METHOD An_unrecognized_version_is_reported_once_with_its_owner
TEST('An_unrecognized_version_is_reported_once_with_its_owner');
_M_Arm();
_M_TakeLoss();
_version := 7;                            // a real image, written by another layout
AssertFalse(Condition := _u.Child.M_RestoreStationCfg(pVersion := ADR(_version),
    SchemaVersion := 1),
    Message := 'an unrecognized image is REJECTED, never read by field position');
AssertEquals_UINT(Expected := 1, Actual := _version,
    Message := 'the version is stamped forward so the loss annunciates once, not every boot');
AssertTrue(Condition := _M_TakeLoss(),
    Message := 'losing a real image is reported (3.8b: never silent)');
AssertEquals_STRING(Expected := 'Test.Durability.Child', Actual := _path,
    Message := 'the report names the OWNING module, which is what makes it actionable');
AssertEquals_UINT(Expected := 1, Actual := _expected,
    Message := 'the report carries the schema this build understands');
AssertEquals_UINT(Expected := 7, Actual := _found,
    Message := 'and the schema actually found');
AssertFalse(Condition := _M_TakeLoss(),
    Message := 'taking a loss clears it: one annunciation per boot, not one per scan');
TEST_FINISHED();
END_METHOD

// §3.8b: the annunciation is AUTO_RESET and therefore never blocking. The
// consequence belongs to E_ConfigRestorePolicy, so a station that declared
// DEFAULTS_AND_ANNUNCIATE really does keep running while the alarm stands.
METHOD The_root_annunciates_a_loss_without_blocking_on_its_own
TEST('The_root_annunciates_a_loss_without_blocking_on_its_own');
_M_Arm();
_M_TakeLoss();
_u.SetConfigRestorePolicy(Policy := E_ConfigRestorePolicy.DEFAULTS_AND_ANNUNCIATE);
_version := 9;
_u.Child.M_RestoreStationCfg(pVersion := ADR(_version), SchemaVersion := 1);
_u();                                     // OnCyclic drains and annunciates
AssertTrue(Condition := _u.ConfigPersist.RestoreLost,
    Message := 'the root publishes that something in its subtree lost its image');
AssertEquals_STRING(Expected := 'Test.Durability.Child',
    Actual := _u.ConfigPersist.LostPath,
    Message := 'and publishes whose');
AssertFalse(Condition := _u.ConfigPersist.RestoreAcknowledged,
    Message := 'nobody has accepted the loss yet');
AssertFalse(Condition := _u.AlarmLog.Blocking,
    Message := 'the standing annunciation is AUTO_RESET: loud, never a Start block');
_released := _u.ReleaseReportStart(Report := _report);
AssertTrue(Condition := _released,
    Message := 'DEFAULTS_AND_ANNUNCIATE runs the station and lets the alarm stand');
TEST_FINISHED();
END_METHOD

// §3.8b BLOCK_UNTIL_ACKNOWLEDGED: no START_STOP release until an operator of at
// least ENGINEER level accepts the loss. The release is restored by the
// ACKNOWLEDGEMENT, never by the loss going away - nothing brings a lost image back.
METHOD Blocking_policy_refuses_start_until_an_engineer_acknowledges
TEST('Blocking_policy_refuses_start_until_an_engineer_acknowledges');
_M_Arm();
_M_TakeLoss();
_u.SetConfigRestorePolicy(Policy := E_ConfigRestorePolicy.BLOCK_UNTIL_ACKNOWLEDGED);
_version := 11;
_u.Child.M_RestoreStationCfg(pVersion := ADR(_version), SchemaVersion := 1);
_u();
AssertTrue(Condition := _u.ConfigPersist.RestoreLost,
    Message := 'the loss is published');
_released := _u.ReleaseReportStart(Report := _report);
AssertFalse(Condition := _released,
    Message := 'a station that lost its commissioning does not start pretending it did not');
AssertFalse(Condition := _u.Start(),
    Message := 'and Start consumes that same report, so the two cannot disagree');
// An operator below ENGINEER cannot make this go away. A login or logout is a
// REQUEST that Access.Cyclic applies on the Unit's next call, so each is followed
// by one - without it the level asserted against was simply the previous one.
_u.Access.RequestLogout();
_u();
AssertFalse(Condition := _u.AcknowledgeConfigRestore(),
    Message := 'acknowledging a lost commissioning is an ENGINEER-level act (3.8b)');
AssertFalse(Condition := _u.ConfigPersist.RestoreAcknowledged,
    Message := 'a refused acknowledgement changes nothing');
AssertTrue(Condition := _u.Access.RequestLogin(User := 'eng', Secret := '4242'),
    Message := 'the fixture provides an ENGINEER session');
_u();
AssertTrue(Condition := _u.AcknowledgeConfigRestore(),
    Message := 'an ENGINEER may accept the loss');
_released := _u.ReleaseReportStart(Report := _report);
AssertTrue(Condition := _released,
    Message := 'the acknowledgement, not the condition, is what releases Start again');
AssertTrue(Condition := _u.ConfigPersist.RestoreLost,
    Message := 'and the loss itself is still published: acknowledged is not undone');
_u.Access.RequestLogout();
_u.SetConfigRestorePolicy(Policy := E_ConfigRestorePolicy.DEFAULTS_AND_ANNUNCIATE);
TEST_FINISHED();
END_METHOD

// §3.8b: "Transport acknowledgement and Accepted mean a value is LIVE, not that
// it is DURABLE." This is that sentence as a test.
METHOD An_accepted_write_is_pending_until_the_store_completes
TEST('An_accepted_write_is_pending_until_the_store_completes');
_M_Arm();
_u.SetConfigPersistWindow(WindowMs := 60000);
_persist.M_SetOutcome(Failed := FALSE, Refuse := FALSE);
_persist.M_SetHold(Hold := TRUE);         // the store does not finish yet
AssertTrue(Condition := _u.WriteConfig(TargetPath := 'Test.Durability',
    WriteKey := 'probe.cycleLimit', Revision := 1, TextValue := '42'),
    Message := 'the write is accepted');
AssertTrue(Condition := _u.ConfigPersist.Pending,
    Message := 'accepted means LIVE - the root publishes that it is not yet durable');
AssertFalse(Condition := _u.ConfigPersist.Failed,
    Message := 'pending is not failed');
_u();
AssertTrue(Condition := _u.ConfigPersist.Pending,
    Message := 'and it stays pending for as long as the store is still working');
_persist.M_SetHold(Hold := FALSE);
_u();
_u();
AssertFalse(Condition := _u.ConfigPersist.Pending,
    Message := 'the value is durable once the store completes');
AssertFalse(Condition := _u.ConfigPersist.Failed,
    Message := 'a completed write is not a failed one');
TEST_FINISHED();
END_METHOD

METHOD A_store_that_refuses_publishes_PersistFailed
TEST('A_store_that_refuses_publishes_PersistFailed');
_M_Arm();
_u.SetConfigPersistWindow(WindowMs := 60000);
_persist.M_SetHold(Hold := FALSE);
_persist.M_SetOutcome(Failed := FALSE, Refuse := TRUE);
AssertTrue(Condition := _u.WriteConfig(TargetPath := 'Test.Durability',
    WriteKey := 'probe.cycleLimit', Revision := 1, TextValue := '43'),
    Message := 'the VALUE is still accepted: it is live, and that is not in doubt');
AssertTrue(Condition := _u.ConfigPersist.Failed,
    Message := 'a store that will not even start is a failure, not a quiet no-op');
AssertTrue(Condition := _u.ConfigPersist.Pending,
    Message := 'and the value is STILL not durable, so it stays pending');
AssertFalse(Condition := _u.AlarmLog.Blocking,
    Message := 'the annunciation does not stop a machine that can still finish its parts');
// A store that starts working again clears both on the next accepted write.
_persist.M_SetOutcome(Failed := FALSE, Refuse := FALSE);
AssertTrue(Condition := _u.WriteConfig(TargetPath := 'Test.Durability',
    WriteKey := 'probe.cycleLimit', Revision := 1, TextValue := '44'),
    Message := 'a later write is accepted');
_u();
_u();
AssertFalse(Condition := _u.ConfigPersist.Failed,
    Message := 'a successful write clears the failure it re-armed');
TEST_FINISHED();
END_METHOD

// §3.8b declares a BOUNDED window, and a bound nobody measures is not a bound.
// WindowMs := 0 declares "durable in the same scan or not at all", which is the
// honest declaration for a store that cannot be slow.
METHOD An_elapsed_window_publishes_PersistFailed
TEST('An_elapsed_window_publishes_PersistFailed');
_M_Arm();
IF NOT _winArmed THEN
    _winArmed := TRUE;
    _persist.M_SetOutcome(Failed := FALSE, Refuse := FALSE);
    _persist.M_SetHold(Hold := TRUE);     // never completes
    _u.SetConfigPersistWindow(WindowMs := 0);
    AssertTrue(Condition := _u.WriteConfig(TargetPath := 'Test.Durability',
        WriteKey := 'probe.cycleLimit', Revision := 1, TextValue := '45'),
        Message := 'the write is accepted');
    AssertTrue(Condition := _u.ConfigPersist.Pending, Message := 'and is pending');
    RETURN;                               // the window is measured in TIME(), which
END_IF                                    // does not advance inside one scan
_u();
_winScans := _winScans + 1;
IF NOT _u.ConfigPersist.Failed AND (_winScans < 50) THEN
    RETURN;                               // bounded: 50 scans, far past a 0 ms window
END_IF
AssertTrue(Condition := _u.ConfigPersist.Failed,
    Message := 'a store still working past the DECLARED window has failed the declaration');
AssertTrue(Condition := _u.ConfigPersist.Pending,
    Message := 'the value is still not durable, so it is still pending');
_persist.M_SetHold(Hold := FALSE);
_u.SetConfigPersistWindow(WindowMs := PL_Fraktal.CONFIG_PERSIST_WINDOW_MS);
_u();
TEST_FINISHED();
END_METHOD

END_FUNCTION_BLOCK

// ---- Fraktal_Tests/FB_ConfigSet_Tests.TcPOU
// Core §3.8b under test, the half that is about CONTENT:
//
//   * a set is a PROJECTION of the same deterministic walk that builds the
//     §3.10.2 manifest - not a second list of what a station's configuration
//     consists of, which would be free to drift from the first;
//   * it is records keyed by (Scope, WriteKey), never a byte image, which is
//     what lets one bad value be rejected without rejecting all of them;
//   * a load is STAGED and ALL-OR-NOTHING, so a set that is wrong anywhere
//     changes nothing anywhere;
//   * and the whole set moves as TEXT, because a set that cannot leave the
//     controller is just retentive memory with a name on it.
FUNCTION_BLOCK FB_ConfigSet_Tests EXTENDS TcUnit.FB_TestSuite
VAR
    _u       : FB_ProbeConfigUnit;
    _init    : BOOL;
    // PL_Fraktal.MAX_CONFIG_SETS is 4 and the store never evicts a set, so every
    // DELIBERATELY WRONG import shares the one name 'imported' (each overwrites
    // the last). Seven distinct names filled the store by the fifth test, and the
    // later imports were refused as 'full' before reaching the rule they test.
    _store   : FB_LocalConfigStore;
    _json    : FB_ConfigSetJson;
    _pager   : FB_ConfigPager;
    _page    : ST_ConfigPage;
    _info    : ST_ConfigSetInfo;
    _record  : ST_ConfigRecord;
    _decoded : ST_ConfigRecord;
    _line    : STRING(480);
    _i       : INT;
    _capabilities : INT;
    // A whole Unit is far too large for a method local: as one it put ~330 KB on a
    // 48 KB task stack (C0297) and the suite could never run. It lives here instead.
    _bare     : FB_ProbeConfigUnit;
    _bareInit : BOOL;
END_VAR

A_saved_set_is_the_manifest_walk_projected();
A_set_round_trips_through_the_store();
Loading_a_set_restores_every_value_it_carries();
One_bad_record_aborts_the_whole_load_and_names_it();
A_capability_that_no_longer_exists_is_reported_not_dropped();
A_set_from_another_root_is_refused();
A_record_round_trips_through_its_json_line();
A_malformed_json_line_is_refused_whole();
A_model_set_is_not_applied_as_per_field_writes();
Set_operations_need_a_store_and_the_CONFIG_SET_gate();
A_deleted_set_is_gone_and_frees_its_slot();
A_line_longer_than_a_request_imports_in_pieces();

// One-time wiring. Nothing here is persistence-specific: a store is injected
// exactly as a composition root injects it, and every value in the resulting
// sets came from an ordinary M_RegisterConfig* call on the probes.
METHOD PRIVATE _M_Arm
IF _init THEN
    RETURN;
END_IF
_init := TRUE;
_u.Setup(Name := 'Test.CfgSet');
_u();
_u.SetConfigStore(Store := _store);
// The store is PERSISTENT, so it still holds whatever the previous run saved:
// start every run from an empty store, through the same delete a station has.
FOR _i := 1 TO PL_Fraktal.MAX_CONFIG_SETS DO
    IF NOT _store.M_InfoAt(Index := 1, Info := _info) THEN
        EXIT;
    END_IF
    _u.DeleteConfigSet(SetName := _info.SetName);
END_FOR
END_METHOD

// Count the writable STATION_CFG capabilities the MANIFEST publishes, by walking
// it exactly as a client does. The set has to contain the same number - that
// equality is what "a set is a projection of the same walk" means in practice.
METHOD PRIVATE _M_CountStationCapabilities : INT
VAR
    page  : INT;
    i     : INT;
    pages : INT;
END_VAR
_M_CountStationCapabilities := 0;
pages := 1;
FOR page := 0 TO 63 DO
    IF page >= pages THEN
        RETURN;
    END_IF
    _pager.M_Setup(Target := ADR(_page), PageIndex := page, Revision := 1);
    _u.M_AppendConfig(Pager := _pager);
    _pager.M_Finish();
    pages := _page.PageCount;
    FOR i := 1 TO _page.EntryCount DO
        IF _page.Entries[i].Writable THEN
            IF _page.Entries[i].ConfigKind = E_ConfigKind.STATION_CFG THEN
                _M_CountStationCapabilities := _M_CountStationCapabilities + 1;
            END_IF
        END_IF
    END_FOR
END_FOR
END_METHOD

// Push one JSON line into the store through the ordinary import route, so a
// suite can build a DELIBERATELY WRONG set the same way a foreign tool would.
METHOD PRIVATE _M_Import : BOOL
VAR_INPUT
    Line   : STRING(480);
    Commit : BOOL;
END_VAR
_M_Import := _u.ImportConfigSetLine(Line := Line, Commit := Commit);
END_METHOD

METHOD A_saved_set_is_the_manifest_walk_projected
TEST('A_saved_set_is_the_manifest_walk_projected');
_M_Arm();
_capabilities := _M_CountStationCapabilities();
AssertTrue(Condition := _capabilities > 0,
    Message := 'the fixture publishes STATION_CFG capabilities to project');
AssertTrue(Condition := _u.SaveConfigSet(SetName := 'baseline',
    Kind := E_ConfigKind.STATION_CFG),
    Message := 'a station set saves');
AssertTrue(Condition := _store.M_ReadInfo(SetName := 'baseline', Info := _info),
    Message := 'and is readable back out of the store');
AssertEquals_INT(Expected := _capabilities, Actual := _info.RecordCount,
    Message := 'the set contains exactly the capabilities the manifest publishes - one walk, not two');
AssertEquals_STRING(Expected := 'Test.CfgSet', Actual := _info.RootIdentity,
    Message := 'a set carries the identity of the root that produced it');
AssertTrue(Condition := _info.ConfigRev > 0,
    Message := 'and the ConfigRev it was taken at');
TEST_FINISHED();
END_METHOD

METHOD A_set_round_trips_through_the_store
TEST('A_set_round_trips_through_the_store');
_M_Arm();
_u.SaveConfigSet(SetName := 'baseline', Kind := E_ConfigKind.STATION_CFG);
AssertTrue(Condition := _store.M_ReadInfo(SetName := 'baseline', Info := _info),
    Message := 'the header reads back');
AssertTrue(Condition := _store.M_ReadRecord(SetName := 'baseline', Index := 1,
    Record := _record), Message := 'and so does record 1');
AssertTrue(Condition := _record.WriteKey <> '',
    Message := 'every record carries the mutation identity it will be replayed through');
AssertFalse(Condition := _store.M_ReadRecord(SetName := 'baseline',
    Index := _info.RecordCount + 1, Record := _record),
    Message := 'reading past the end is refused, not clamped');
AssertFalse(Condition := _store.M_ReadInfo(SetName := 'nosuchset', Info := _info),
    Message := 'an absent set is absent, not empty');
AssertTrue(Condition := _u.ListConfigSets(),
    Message := 'the listing is served');
AssertTrue(Condition := _u.ConfigSetCount >= 1,
    Message := 'and shows the set that was just saved');
TEST_FINISHED();
END_METHOD

METHOD Loading_a_set_restores_every_value_it_carries
TEST('Loading_a_set_restores_every_value_it_carries');
_M_Arm();
_u.WriteConfig(TargetPath := 'Test.CfgSet', WriteKey := 'probe.cycleLimit',
    Revision := 1, TextValue := '250');
AssertTrue(Condition := _u.SaveConfigSet(SetName := 'commissioned',
    Kind := E_ConfigKind.STATION_CFG), Message := 'save the commissioned state');
// Somebody then changes the machine.
_u.WriteConfig(TargetPath := 'Test.CfgSet', WriteKey := 'probe.cycleLimit',
    Revision := 1, TextValue := '7');
AssertEquals_DINT(Expected := 7, Actual := _u.CycleLimit,
    Message := 'the live value really changed');
AssertTrue(Condition := _u.LoadConfigSet(SetName := 'commissioned'),
    Message := 'the saved set loads');
AssertEquals_DINT(Expected := 250, Actual := _u.CycleLimit,
    Message := 'and the commissioned value is back, replayed through the owning handler');
TEST_FINISHED();
END_METHOD

// §3.8b: "one rejection aborts the whole load naming the offending
// (Scope, WriteKey)" and "a half-applied machine parametrization is never a
// valid outcome". The set below is valid in every record but one.
METHOD One_bad_record_aborts_the_whole_load_and_names_it
TEST('One_bad_record_aborts_the_whole_load_and_names_it');
_M_Arm();
_u.WriteConfig(TargetPath := 'Test.CfgSet', WriteKey := 'probe.cycleLimit',
    Revision := 1, TextValue := '99');
// A set whose FIRST record is fine and whose SECOND is out of the declared
// range - built as text, exactly as a foreign tool or a hand edit would.
AssertTrue(Condition := _M_Import(Line :=
    '{"set":"imported","root":"Test.CfgSet","schema":1,"configRev":1,"kind":1,"model":"","records":2,"created":0,"clock":0}',
    Commit := FALSE), Message := 'the header opens the import');
AssertTrue(Condition := _M_Import(Line :=
    '{"scope":"Test.CfgSet.Child","key":"probe.retries","rev":1,"kind":1,"type":0,"value":"4"}',
    Commit := FALSE), Message := 'a good record is taken');
AssertTrue(Condition := _M_Import(Line :=
    '{"scope":"Test.CfgSet","key":"probe.cycleLimit","rev":1,"kind":1,"type":0,"value":"99999"}',
    Commit := TRUE), Message := 'and so is the out-of-range one: the STORE does not validate');
AssertFalse(Condition := _u.LoadConfigSet(SetName := 'imported'),
    Message := 'the LOAD validates, and one bad record refuses the whole set');
AssertEquals_DINT(Expected := 99, Actual := _u.CycleLimit,
    Message := 'nothing was applied - not even the record that came BEFORE the bad one');
AssertEquals_DINT(Expected := 3, Actual := _u.Child.Retries,
    Message := 'and not the good record in another module either');
AssertEquals_STRING(Expected := 'Test.CfgSet',
    Actual := _u.ConfigPersist.LastRejectScope,
    Message := 'the refusal names the scope of the offending record');
AssertEquals_STRING(Expected := 'probe.cycleLimit',
    Actual := _u.ConfigPersist.LastRejectKey,
    Message := 'and its write key');
TEST_FINISHED();
END_METHOD

// §3.8b: "Records whose capability no longer exists in the target are reported,
// never silently dropped." A set that quietly skipped the one value that
// mattered would restore a machine to ALMOST its commissioned state, which is
// the failure that is hardest to notice.
METHOD A_capability_that_no_longer_exists_is_reported_not_dropped
TEST('A_capability_that_no_longer_exists_is_reported_not_dropped');
_M_Arm();
_M_Import(Line :=
    '{"set":"imported","root":"Test.CfgSet","schema":1,"configRev":1,"kind":1,"model":"","records":1,"created":0,"clock":0}',
    Commit := FALSE);
_M_Import(Line :=
    '{"scope":"Test.CfgSet","key":"probe.valueThatWasRemoved","rev":1,"kind":1,"type":0,"value":"1"}',
    Commit := TRUE);
AssertFalse(Condition := _u.LoadConfigSet(SetName := 'imported'),
    Message := 'a record nothing owns any more refuses the load');
AssertEquals_STRING(Expected := 'probe.valueThatWasRemoved',
    Actual := _u.ConfigPersist.LastRejectKey,
    Message := 'and is REPORTED by name rather than passed over');
TEST_FINISHED();
END_METHOD

METHOD A_set_from_another_root_is_refused
TEST('A_set_from_another_root_is_refused');
_M_Arm();
_M_Import(Line :=
    '{"set":"imported","root":"SomeOtherPress","schema":1,"configRev":1,"kind":1,"model":"","records":1,"created":0,"clock":0}',
    Commit := FALSE);
_M_Import(Line :=
    '{"scope":"SomeOtherPress","key":"probe.cycleLimit","rev":1,"kind":1,"type":0,"value":"5"}',
    Commit := TRUE);
AssertFalse(Condition := _u.LoadConfigSet(SetName := 'imported'),
    Message := 'a set carries the identity of the root that produced it so this can be asked');
AssertEquals_STRING(Expected := 'SomeOtherPress',
    Actual := _u.ConfigPersist.LastRejectScope,
    Message := 'and the refusal names the root it actually came from');
TEST_FINISHED();
END_METHOD

// A set that cannot leave the controller is retentive memory with a name on it.
// One JSON object per record is what makes it movable - and keeps every value
// independently identified and independently rejectable, which is exactly the
// property §3.8b says a byte image loses.
METHOD A_record_round_trips_through_its_json_line
TEST('A_record_round_trips_through_its_json_line');
_M_Arm();
_record.Scope := 'Test.CfgSet.Child';
_record.WriteKey := 'probe.label';
_record.Revision := 2;
_record.Kind := E_ConfigKind.STATION_CFG;
_record.ValueType := E_ConfigValueType.TEXT;
_record.ValueText := 'a "quoted" value';   // the two characters JSON must escape
_line := _json.M_Record(Record := _record);
AssertTrue(Condition := _line <> '',
    Message := 'a valid record renders');
AssertTrue(Condition := _json.M_ParseRecord(Line := _line, Record := _decoded),
    Message := 'and parses back');
AssertEquals_STRING(Expected := 'Test.CfgSet.Child', Actual := _decoded.Scope,
    Message := 'the owning scope survives the round trip');
AssertEquals_STRING(Expected := 'probe.label', Actual := _decoded.WriteKey,
    Message := 'so does the mutation identity');
AssertEquals_STRING(Expected := 'a "quoted" value', Actual := _decoded.ValueText,
    Message := 'and so does a value containing the delimiter itself');
AssertEquals_UDINT(Expected := 2, Actual := _decoded.Revision,
    Message := 'the capability revision travels with the record, so a load can reject a value whose meaning changed');
TEST_FINISHED();
END_METHOD

METHOD A_malformed_json_line_is_refused_whole
TEST('A_malformed_json_line_is_refused_whole');
_M_Arm();
_decoded.WriteKey := 'untouched';
AssertFalse(Condition := _json.M_ParseRecord(
    Line := '{"scope":"x","key":"y","rev":1,"kind":1,"type":0', Record := _decoded),
    Message := 'a truncated line is not a record');
AssertFalse(Condition := _json.M_ParseRecord(
    Line := '{"scope":"x","key":"y","rev":"notanumber","kind":1,"type":0,"value":"1"}',
    Record := _decoded), Message := 'nor is one whose revision is not a number');
AssertFalse(Condition := _json.M_ParseRecord(
    Line := '{"scope":"x","key":"y","rev":1,"kind":9,"type":0,"value":"1"}',
    Record := _decoded), Message := 'nor one whose kind is outside E_ConfigKind');
AssertEquals_STRING(Expected := 'untouched', Actual := _decoded.WriteKey,
    Message := 'a refused line leaves the caller record exactly as it was');
AssertFalse(Condition := _json.M_ParseHeader(
    Line := '{"scope":"x","key":"y","rev":1,"kind":1,"type":0,"value":"1"}',
    Info := _info), Message := 'a record line is not a header, and says so');
TEST_FINISHED();
END_METHOD

// §3.8b: a MODEL set "shall be applied through the §3.8 changeover transaction
// ... never as a sequence of per-field writes". Replaying it here would be
// exactly that forbidden sequence, so it is refused. Saving one is supported;
// loading one is a changeover this build does not implement, and refusing is
// the honest half of that.
METHOD A_model_set_is_not_applied_as_per_field_writes
TEST('A_model_set_is_not_applied_as_per_field_writes');
_M_Arm();
_M_Import(Line :=
    '{"set":"imported","root":"Test.CfgSet","schema":1,"configRev":1,"kind":0,"model":"ALU","records":1,"created":0,"clock":0}',
    Commit := FALSE);
_M_Import(Line :=
    '{"scope":"Test.CfgSet","key":"probe.cycleLimit","rev":1,"kind":0,"type":0,"value":"12"}',
    Commit := TRUE);
AssertFalse(Condition := _u.LoadConfigSet(SetName := 'imported'),
    Message := 'a model set is not replayed as per-field writes');
AssertEquals_STRING(Expected := 'ALU', Actual := _u.ConfigPersist.LastRejectScope,
    Message := 'and the refusal names the model it was for');
TEST_FINISHED();
END_METHOD

// §3.8b/§7.7: saving, loading or importing a SET is the separate gated action
// CONFIG_SET, "because replacing a machine's entire parametrization is not the
// same decision as changing one number". And a root with no store offers the
// operations not at all rather than failing when somebody finally tries.
METHOD Set_operations_need_a_store_and_the_CONFIG_SET_gate
TEST('Set_operations_need_a_store_and_the_CONFIG_SET_gate');
_M_Arm();
IF NOT _bareInit THEN
    _bareInit := TRUE;
    _bare.Setup(Name := 'Test.NoStore');   // registers once, like any root
END_IF
_bare();
AssertFalse(Condition := _bare.ConfigPersist.StorePresent,
    Message := 'a root with no store says so, rather than pretending');
AssertFalse(Condition := _bare.SaveConfigSet(SetName := 'x',
    Kind := E_ConfigKind.STATION_CFG),
    Message := 'and refuses to save');
AssertFalse(Condition := _bare.LoadConfigSet(SetName := 'x'),
    Message := 'and to load');
AssertTrue(Condition := _u.ConfigPersist.StorePresent,
    Message := 'a wired root publishes that sets are available');
AssertEquals_DINT(Expected := TO_DINT(E_ConfigStore.LOCAL_RETAIN),
    Actual := TO_DINT(_u.ConfigPersist.StoreKind),
    Message := 'and publishes WHERE they live, so a saved set is not taken on faith');
AssertTrue(Condition := _u.Access.RequestLogout(),
    Message := 'no session is required by the shipped fully-open policy');
AssertTrue(Condition := _u.SaveConfigSet(SetName := 'open',
    Kind := E_ConfigKind.STATION_CFG),
    Message := 'so an open station saves without a login - access control is never a silent lock-in');
TEST_FINISHED();
END_METHOD

// §3.8b round trip. An exported line may hold 480 characters but a request
// carries 255, so a long record arrives in pieces (IMPORT_CONFIG_SET with
// IntValue = 1). Without the join, a station's own export could not come back.
METHOD A_line_longer_than_a_request_imports_in_pieces
VAR
    header : STRING(480);
    first  : STRING(255);
    rest   : STRING(255);
    k      : INT;
    size   : INT;                          // measured by scanning, not by LEN
    p      : POINTER TO BYTE;
END_VAR
TEST('A_line_longer_than_a_request_imports_in_pieces');
_M_Arm();
// The previous test leaves the store full: free a slot, then reuse fill2's
// header so the import overwrites a set this suite owns.
_u.DeleteConfigSet(SetName := 'fill1');
_u.ExportConfigSetLine(SetName := 'fill2', Line := 0);
header := _u.ConfigSetDocument;
AssertTrue(Condition := header <> '', Message := 'a header to import under');
_record.Scope := 'Test.CfgSet.Child.Long';
_record.WriteKey := '';
FOR k := 1 TO 14 DO
    _record.WriteKey := CONCAT(_record.WriteKey, 'probe.long');
END_FOR
_record.Revision := 1;
_record.Kind := E_ConfigKind.STATION_CFG;
_record.ValueType := E_ConfigValueType.TEXT;
_record.ValueText := '';
FOR k := 1 TO 7 DO
    _record.ValueText := CONCAT(_record.ValueText, '0123456789');
END_FOR
_line := _json.M_Record(Record := _record);
// The length is measured by scanning to the terminator, independently of LEN:
// the standard string functions are specified to 255 characters, so neither
// LEN nor CONCAT may be trusted past it without proof.
size := 0;
p := ADR(_line);
WHILE size < 480 AND p^ <> 0 DO
    size := size + 1;
    p := p + 1;
END_WHILE
AssertTrue(Condition := size > 255,
    Message := CONCAT('the record renders past 255 characters; scanned ', INT_TO_STRING(size)));
// Measured on the runtime (2026-09-28): LEN reported 255 for this 290-character
// line. That is why the codec scans instead, and why this test does too.
AssertTrue(Condition := _json.M_ParseRecord(Line := _line, Record := _decoded),
    Message := 'the long line is whole: it parses back');
AssertEquals_STRING(Expected := _record.ValueText, Actual := _decoded.ValueText,
    Message := 'and its value is intact, so rendering did not truncate');
// Pieces by byte copy, so the test does not depend on LEFT/MID past 255.
MEMSET(ADR(first), 0, SIZEOF(first));
MEMSET(ADR(rest), 0, SIZEOF(rest));
MEMCPY(ADR(first), ADR(_line), 200);
IF size > 200 THEN
    MEMCPY(ADR(rest), ADR(_line) + 200, TO_UDINT(MIN(size - 200, 255)));
END_IF
AssertTrue(Condition := _M_Import(Line := header, Commit := FALSE),
    Message := 'the header opens the import');
AssertTrue(Condition := _u.ImportConfigSetPiece(Piece := first, More := TRUE,
    Commit := FALSE), Message := 'the first piece is held');
AssertTrue(Condition := _u.ImportConfigSetPiece(Piece := rest, More := FALSE,
    Commit := TRUE), Message := 'the last piece completes the line, which imports and commits');
AssertTrue(Condition := _store.M_ReadRecord(SetName := 'fill2', Index := 1,
    Record := _decoded), Message := 'the joined record is in the store');
AssertEquals_STRING(Expected := _record.ValueText, Actual := _decoded.ValueText,
    Message := 'and its value arrived whole, not truncated at 255');
AssertEquals_STRING(Expected := _record.WriteKey, Actual := _decoded.WriteKey,
    Message := 'as did its 140-character key');
// Refused, never truncated: pieces that would exceed the line width.
AssertTrue(Condition := _u.ImportConfigSetPiece(Piece := first, More := TRUE,
    Commit := FALSE), Message := 'a piece is held');
AssertTrue(Condition := _u.ImportConfigSetPiece(Piece := first, More := TRUE,
    Commit := FALSE), Message := 'and a second (400 characters so far)');
AssertFalse(Condition := _u.ImportConfigSetPiece(Piece := first, More := FALSE,
    Commit := FALSE), Message := 'a join past 480 characters is refused');
TEST_FINISHED();
END_METHOD

// §3.8b: without a delete, a store that has held MAX_CONFIG_SETS names can
// only ever overwrite one of them again - a new product's recipe could not be
// kept without destroying an old one under its name.
METHOD A_deleted_set_is_gone_and_frees_its_slot
VAR
    fill : STRING(80);
END_VAR
TEST('A_deleted_set_is_gone_and_frees_its_slot');
_M_Arm();
// The earlier tests leave the store full, so start from empty: this test is
// about what delete does, not about which sets happened to be there.
FOR _i := 1 TO PL_Fraktal.MAX_CONFIG_SETS DO
    IF NOT _store.M_InfoAt(Index := 1, Info := _info) THEN
        EXIT;
    END_IF
    _u.DeleteConfigSet(SetName := _info.SetName);
END_FOR
AssertTrue(Condition := _u.SaveConfigSet(SetName := 'scratch',
    Kind := E_ConfigKind.STATION_CFG), Message := 'a set to delete is saved');
AssertTrue(Condition := _u.DeleteConfigSet(SetName := 'scratch'),
    Message := 'an existing set is deleted');
AssertFalse(Condition := _store.M_ReadInfo(SetName := 'scratch', Info := _info),
    Message := 'and is no longer readable');
AssertFalse(Condition := _u.DeleteConfigSet(SetName := 'scratch'),
    Message := 'deleting what is not there is refused, not silently accepted');
AssertTrue(Condition := _u.ConfigPersist.Pending,
    Message := 'a delete changes retained memory, so it is not durable until written out');
AssertEquals_INT(Expected := 0, Actual := _store.M_Count(),
    Message := 'every set can be removed');
// The freed slots are usable: fill the store to capacity under fresh names.
FOR _i := 1 TO PL_Fraktal.MAX_CONFIG_SETS DO
    fill := CONCAT('fill', INT_TO_STRING(_i));
    AssertTrue(Condition := _u.SaveConfigSet(SetName := fill,
        Kind := E_ConfigKind.STATION_CFG), Message := 'each freed slot takes a new name');
END_FOR
TEST_FINISHED();
END_METHOD

END_FUNCTION_BLOCK

// ---- Fraktal_Tests/FB_DataClass_Tests.TcPOU
// Core §3.8d under test: data classes and raise-only per-value access.
// Every test body is guarded: TcUnit calls finished tests every scan, and these
// write to one shared probe.
FUNCTION_BLOCK FB_DataClass_Tests EXTENDS TcUnit.FB_TestSuite
VAR
    _u     : FB_ProbeConfigUnit;
    _users : FB_LocalAccessProvider;
    _store : FB_LocalConfigStore;
    _pager : FB_ConfigPager;
    _page  : ST_ConfigPage;
    _entry : ST_ConfigEntry;
    _info  : ST_ConfigSetInfo;
    _init  : BOOL;
    _i     : INT;
    _w1, _w2, _w3, _w4, _w5, _w6, _w7 : BOOL;
END_VAR

Builtin_class_uses_DATA_WRITE();
A_public_class_lets_an_operator_edit_its_values();
A_value_can_only_raise_its_class();
An_undeclared_class_fails_closed();
Declaring_a_class_again_keeps_an_edited_level();
The_manifest_publishes_effective_levels();
A_set_load_needs_the_write_level_of_every_record();

// One-time wiring through the surface a composition root uses.
METHOD PRIVATE _M_Arm
IF _init THEN
    RETURN;
END_IF
_init := TRUE;
_u.Setup(Name := 'Test.Class');
_u();
// Not under test here: a volatile table, so no previous run's file is a precondition.
_users.M_UseKey(Key := '');
_users.Register(User := 'op', Pin := '1111', Level := E_AccessLevel.OPERATOR);
_users.Register(User := 'eng', Pin := '4242', Level := E_AccessLevel.ENGINEER);
_users.Register(User := 'adm', Pin := '9999', Level := E_AccessLevel.ADMIN);
_u.Access.Setup(Provider := _users, pAlarmLog := ADR(_u.AlarmLog));
_u.Access.ConfigureRequired(Gate := E_GatedAction.DATA_WRITE, Level := E_AccessLevel.ENGINEER);
_u.Access.ConfigureRequired(Gate := E_GatedAction.DATA_READ, Level := E_AccessLevel.NONE);
_u.M_DeclareDataClass(ClassId := 'public', LabelKey := 'project.dataClass.public',
    ReadLevel := E_AccessLevel.NONE, WriteLevel := E_AccessLevel.OPERATOR);
// The class table is PERSISTENT: undo whatever a previous, interrupted run edited.
_u.Access.M_SetClassLevel(ClassId := 'public', Level := E_AccessLevel.OPERATOR, ForWrite := TRUE);
_u.Access.M_SetClassLevel(ClassId := 'public', Level := E_AccessLevel.NONE, ForWrite := FALSE);
_u.Child.M_SetConfigAccess(WriteKey := 'probe.retries', ClassId := 'public',
    MinReadLevel := E_AccessLevel.NONE, MinWriteLevel := E_AccessLevel.NONE);
_u.Child.M_SetConfigAccess(WriteKey := 'probe.enabled', ClassId := 'public',
    MinReadLevel := E_AccessLevel.NONE, MinWriteLevel := E_AccessLevel.ENGINEER);
_u.Child.M_SetConfigAccess(WriteKey := 'probe.label', ClassId := 'ghost',
    MinReadLevel := E_AccessLevel.NONE, MinWriteLevel := E_AccessLevel.NONE);
_u.SetConfigStore(Store := _store);
FOR _i := 1 TO PL_Fraktal.MAX_CONFIG_SETS DO
    IF NOT _store.M_InfoAt(Index := 1, Info := _info) THEN
        EXIT;
    END_IF
    _u.DeleteConfigSet(SetName := _info.SetName);
END_FOR
END_METHOD

// A login is a REQUEST that Access.Cyclic applies on the Unit's next call.
METHOD PRIVATE _M_Login
VAR_INPUT
    User : STRING(32);
    Pin  : STRING(32);
END_VAR
_u.Access.RequestLogin(User := User, Secret := Pin);
_u();
END_METHOD

METHOD PRIVATE _M_Logout
_u.Access.RequestLogout();
_u();
END_METHOD

// Walk the manifest exactly as QUERY_CONFIG does, with the root's access context,
// and leave the entry for WriteKey in _entry.
METHOD PRIVATE _M_FindEntry : BOOL
VAR_INPUT
    WriteKey : STRING(160);
END_VAR
VAR
    page  : INT;
    i     : INT;
    pages : INT;
END_VAR
_M_FindEntry := FALSE;
pages := 1;
_pager.M_SetAccess(pAccess := ADR(_u.Access));
FOR page := 0 TO 63 DO
    IF page >= pages THEN
        RETURN;
    END_IF
    _pager.M_Setup(Target := ADR(_page), PageIndex := page, Revision := 1);
    _u.M_AppendConfig(Pager := _pager);
    _pager.M_Finish();
    pages := _page.PageCount;
    FOR i := 1 TO _page.EntryCount DO
        IF _page.Entries[i].WriteKey = WriteKey THEN
            _entry := _page.Entries[i];
            _M_FindEntry := TRUE;
            RETURN;
        END_IF
    END_FOR
END_FOR
END_METHOD

// §3.8d(a): a value registered without a class behaves exactly as before.
METHOD Builtin_class_uses_DATA_WRITE
TEST('Builtin_class_uses_DATA_WRITE');
_M_Arm();
IF NOT _w1 THEN
    _M_Login(User := 'op', Pin := '1111');
    AssertFalse(Condition := _u.WriteConfig(TargetPath := 'Test.Class.Child',
        WriteKey := 'probe.settleTime', Revision := 1, TextValue := '100'),
        Message := 'an OPERATOR cannot write a built-in value while DATA_WRITE is ENGINEER');
    _M_Login(User := 'eng', Pin := '4242');
    AssertTrue(Condition := _u.WriteConfig(TargetPath := 'Test.Class.Child',
        WriteKey := 'probe.settleTime', Revision := 1, TextValue := '100'),
        Message := 'an ENGINEER can');
    _M_Logout();
    _w1 := TRUE;
END_IF
TEST_FINISHED();
END_METHOD

// §3.8d(a): the whole point - one class open to an OPERATOR while the rest of
// the station data stays at ENGINEER.
METHOD A_public_class_lets_an_operator_edit_its_values
TEST('A_public_class_lets_an_operator_edit_its_values');
_M_Arm();
IF NOT _w2 THEN
    _M_Login(User := 'op', Pin := '1111');
    AssertTrue(Condition := _u.WriteConfig(TargetPath := 'Test.Class.Child',
        WriteKey := 'probe.retries', Revision := 1, TextValue := '5'),
        Message := 'a value in the public class is writable at OPERATOR');
    AssertEquals_DINT(Expected := 5, Actual := _u.Child.Retries,
        Message := 'and the value really changed');
    _M_Logout();
    _w2 := TRUE;
END_IF
TEST_FINISHED();
END_METHOD

// §3.8d(c): a value's own minimum raises its class's level, never lowers it.
METHOD A_value_can_only_raise_its_class
TEST('A_value_can_only_raise_its_class');
_M_Arm();
IF NOT _w3 THEN
    _M_Login(User := 'op', Pin := '1111');
    AssertFalse(Condition := _u.WriteConfig(TargetPath := 'Test.Class.Child',
        WriteKey := 'probe.enabled', Revision := 1, TextValue := 'FALSE'),
        Message := 'a public-class value with its own ENGINEER minimum refuses an OPERATOR');
    _M_Login(User := 'eng', Pin := '4242');
    AssertTrue(Condition := _u.WriteConfig(TargetPath := 'Test.Class.Child',
        WriteKey := 'probe.enabled', Revision := 1, TextValue := 'FALSE'),
        Message := 'and accepts an ENGINEER');
    AssertTrue(Condition := _u.Child.M_SetConfigAccess(WriteKey := 'probe.enabled',
        ClassId := 'public', MinReadLevel := E_AccessLevel.NONE, MinWriteLevel := E_AccessLevel.NONE),
        Message := 'the minimum can be taken away again by the code that set it');
    AssertEquals_DINT(Expected := TO_DINT(E_AccessLevel.OPERATOR),
        Actual := TO_DINT(_u.Access.M_DataLevel(ClassId := 'public', MinLevel := E_AccessLevel.NONE,
            ForWrite := TRUE)),
        Message := 'a minimum of NONE leaves the class level, it does not lower it');
    _u.Child.M_SetConfigAccess(WriteKey := 'probe.enabled', ClassId := 'public',
        MinReadLevel := E_AccessLevel.NONE, MinWriteLevel := E_AccessLevel.ENGINEER);
    _M_Logout();
    _w3 := TRUE;
END_IF
TEST_FINISHED();
END_METHOD

// §3.8d: a value placed in a class the root never declared is ADMIN-only, so a
// typo in a class id locks a value down instead of opening it.
METHOD An_undeclared_class_fails_closed
TEST('An_undeclared_class_fails_closed');
_M_Arm();
IF NOT _w4 THEN
    _M_Login(User := 'eng', Pin := '4242');
    AssertFalse(Condition := _u.WriteConfig(TargetPath := 'Test.Class.Child',
        WriteKey := 'probe.label', Revision := 2, TextValue := 'x'),
        Message := 'an undeclared class refuses even an ENGINEER');
    AssertEquals_DINT(Expected := TO_DINT(E_AccessLevel.ADMIN),
        Actual := TO_DINT(_u.Access.M_DataLevel(ClassId := 'ghost', MinLevel := E_AccessLevel.NONE,
            ForWrite := TRUE)),
        Message := 'because it resolves to ADMIN');
    _M_Logout();
    _w4 := TRUE;
END_IF
TEST_FINISHED();
END_METHOD

// §3.8d(b): declared levels are defaults. A class is declared on every boot, and a
// level the deployment edited must survive that.
METHOD Declaring_a_class_again_keeps_an_edited_level
TEST('Declaring_a_class_again_keeps_an_edited_level');
_M_Arm();
IF NOT _w5 THEN
    AssertTrue(Condition := _u.SetDataClassLevel(ClassId := 'public',
        Level := TO_DINT(E_AccessLevel.TECHNICIAN), ForWrite := TRUE),
        Message := 'the policy path edits a class level');
    AssertTrue(Condition := _u.M_DeclareDataClass(ClassId := 'public',
        LabelKey := 'project.dataClass.public', ReadLevel := E_AccessLevel.NONE,
        WriteLevel := E_AccessLevel.OPERATOR), Message := 'the class is declared again, as at boot');
    AssertEquals_DINT(Expected := TO_DINT(E_AccessLevel.TECHNICIAN),
        Actual := TO_DINT(_u.Access.M_DataLevel(ClassId := 'public', MinLevel := E_AccessLevel.NONE,
            ForWrite := TRUE)),
        Message := 'and the edited level stands; the declaration was only a default');
    AssertFalse(Condition := _u.SetDataClassLevel(ClassId := 'public', Level := 9, ForWrite := TRUE),
        Message := 'an out-of-range level is refused');
    _u.SetDataClassLevel(ClassId := 'public', Level := TO_DINT(E_AccessLevel.OPERATOR), ForWrite := TRUE);
    _w5 := TRUE;
END_IF
TEST_FINISHED();
END_METHOD

// §3.8d(d): the PLC computes the effective levels, so a client greys from data;
// and an unreadable value is served WITHOUT its value, never silently dropped.
METHOD The_manifest_publishes_effective_levels
TEST('The_manifest_publishes_effective_levels');
_M_Arm();
IF NOT _w6 THEN
    _M_Logout();
    AssertTrue(Condition := _M_FindEntry(WriteKey := 'probe.retries'),
        Message := 'the public value is in the manifest');
    AssertEquals_STRING(Expected := 'public', Actual := _entry.ClassId, Message := 'with its class');
    AssertEquals_DINT(Expected := TO_DINT(E_AccessLevel.OPERATOR), Actual := TO_DINT(_entry.WriteLevel),
        Message := 'and its effective write level');
    AssertTrue(Condition := _M_FindEntry(WriteKey := 'probe.enabled'),
        Message := 'the raised value is in the manifest');
    AssertEquals_DINT(Expected := TO_DINT(E_AccessLevel.ENGINEER), Actual := TO_DINT(_entry.WriteLevel),
        Message := 'at the RAISED level, not the class level');
    AssertTrue(Condition := _M_FindEntry(WriteKey := 'probe.label'),
        Message := 'the undeclared-class value is still listed');
    AssertFalse(Condition := _entry.Readable, Message := 'as unreadable');
    AssertEquals_STRING(Expected := '', Actual := _entry.ValueText,
        Message := 'and without its value');
    _w6 := TRUE;
END_IF
TEST_FINISHED();
END_METHOD

// §3.8d(e): CONFIG_SET alone cannot replace a value the same user could not edit
// one at a time - otherwise a set is a way around every class.
METHOD A_set_load_needs_the_write_level_of_every_record
TEST('A_set_load_needs_the_write_level_of_every_record');
_M_Arm();
IF NOT _w7 THEN
    _M_Login(User := 'eng', Pin := '4242');
    AssertTrue(Condition := _u.SaveConfigSet(SetName := 'classed',
        Kind := E_ConfigKind.STATION_CFG), Message := 'an ENGINEER saves a station set');
    _M_Login(User := 'op', Pin := '1111');
    AssertFalse(Condition := _u.LoadConfigSet(SetName := 'classed'),
        Message := 'an OPERATOR may not load it: it carries ENGINEER-level values');
    AssertTrue(Condition := _u.ConfigPersist.LastRejectKey <> '',
        Message := 'and the refusal names the record that needed more');
    // The set also carries probe.label, whose class was never declared and so is
    // ADMIN-only: an ENGINEER is refused too, and the refusal names that record.
    _M_Login(User := 'eng', Pin := '4242');
    AssertFalse(Condition := _u.LoadConfigSet(SetName := 'classed'),
        Message := 'an ENGINEER may not load a set carrying an ADMIN-only value');
    AssertEquals_STRING(Expected := 'probe.label', Actual := _u.ConfigPersist.LastRejectKey,
        Message := 'and the refusal names exactly that value');
    _M_Login(User := 'adm', Pin := '9999');
    AssertTrue(Condition := _u.LoadConfigSet(SetName := 'classed'),
        Message := 'a session that could edit every value one at a time may load the set');
    _M_Logout();
    _w7 := TRUE;
END_IF
TEST_FINISHED();
END_METHOD

END_FUNCTION_BLOCK

// ---- Fraktal_Tests/FB_ModelData_Tests.TcPOU
// Core §3.8a under test: a root's model data is editable for every model it
// offers. A request names the model by index (0 = the active one); the value is
// served from, and stored in, that model's own record, and saved back to the
// provider. The running recipe is never touched by another model's edit.
FUNCTION_BLOCK FB_ModelData_Tests EXTENDS TcUnit.FB_TestSuite
VAR
    _u     : FB_ProbeModelUnit;
    _users : FB_LocalAccessProvider;
    _recipes : FB_LocalRecipeProvider;
    _rec0, _recA, _recB : ST_ProbeModelParCfg;
    _pager : FB_ConfigPager;
    _page  : ST_ConfigPage;
    _entry : ST_ConfigEntry;
    _init  : BOOL;
    _w1, _w2, _w3, _w4 : BOOL;
END_VAR

Another_model_is_served_and_edited_in_its_own_record();
An_edit_of_the_active_model_is_saved_to_its_record();
An_unknown_model_is_refused();
Another_model_page_holds_only_its_model_data();

METHOD PRIVATE _M_Arm
IF _init THEN
    RETURN;
END_IF
_init := TRUE;
_rec0.Speed := 1;
_recA.Speed := 10;
_recB.Speed := 20;
_recipes.Register(ModelCode := '', RecipeKey := 'ProbeModel', pData := ADR(_rec0), Size := SIZEOF(_rec0));
_recipes.Register(ModelCode := 'A', RecipeKey := 'ProbeModel', pData := ADR(_recA), Size := SIZEOF(_recA));
_recipes.Register(ModelCode := 'B', RecipeKey := 'ProbeModel', pData := ADR(_recB), Size := SIZEOF(_recB));
_u.ParCfg := _rec0;                         // the active model is '' (no changeover yet)
_u.Setup(Name := 'Test.Model', Provider := _recipes);
_u();
// Not under test here: a volatile table, so no previous run's file is a precondition.
_users.M_UseKey(Key := '');
_users.Register(User := 'eng', Pin := '4242', Level := E_AccessLevel.ENGINEER);
_u.Access.Setup(Provider := _users, pAlarmLog := ADR(_u.AlarmLog));
_u.Access.ConfigureRequired(Gate := E_GatedAction.DATA_WRITE, Level := E_AccessLevel.ENGINEER);
_u.Access.ConfigureRequired(Gate := E_GatedAction.DATA_READ, Level := E_AccessLevel.NONE);
_u.Access.RequestLogin(User := 'eng', Secret := '4242');
_u();
END_METHOD

// Walk the manifest for AvailableModels[ModelIndex] and leave WriteKey's entry.
METHOD PRIVATE _M_Find : BOOL
VAR_INPUT
    ModelIndex : UDINT;
    WriteKey   : STRING(160);
END_VAR
VAR
    i : INT;
END_VAR
_M_Find := FALSE;
_pager.M_SetAccess(pAccess := ADR(_u.Access));
_pager.M_Setup(Target := ADR(_page), PageIndex := 0, Revision := 1);
IF NOT _u.M_AppendModelConfig(Pager := _pager, ModelIndex := ModelIndex) THEN
    RETURN;
END_IF
_pager.M_Finish();
FOR i := 1 TO _page.EntryCount DO
    IF _page.Entries[i].WriteKey = WriteKey THEN
        _entry := _page.Entries[i];
        _M_Find := TRUE;
        RETURN;
    END_IF
END_FOR
END_METHOD

METHOD Another_model_is_served_and_edited_in_its_own_record
TEST('Another_model_is_served_and_edited_in_its_own_record');
_M_Arm();
IF NOT _w1 THEN
    AssertTrue(Condition := _M_Find(ModelIndex := 2, WriteKey := 'probe.speed'),
        Message := 'model B is served');
    AssertEquals_STRING(Expected := '20', Actual := _entry.ValueText,
        Message := 'with B$'s own value, not the running one');
    AssertTrue(Condition := _entry.ModelScoped, Message := 'and marked model-scoped');
    AssertTrue(Condition := _u.WriteModelConfig(ModelIndex := 2, TargetPath := 'Test.Model',
        WriteKey := 'probe.speed', Revision := 1, TextValue := '25'),
        Message := 'B$'s value is edited');
    AssertEquals_DINT(Expected := 25, Actual := _recB.Speed,
        Message := 'into B$'s record, through the provider');
    AssertEquals_DINT(Expected := 1, Actual := _u.ParCfg.Speed,
        Message := 'and the running recipe is untouched');
    AssertEquals_DINT(Expected := 10, Actual := _recA.Speed,
        Message := 'as is every other model');
    _w1 := TRUE;
END_IF
TEST_FINISHED();
END_METHOD

METHOD An_edit_of_the_active_model_is_saved_to_its_record
TEST('An_edit_of_the_active_model_is_saved_to_its_record');
_M_Arm();
IF NOT _w2 THEN
    AssertTrue(Condition := _u.WriteModelConfig(ModelIndex := 0, TargetPath := 'Test.Model',
        WriteKey := 'probe.speed', Revision := 1, TextValue := '7'),
        Message := 'the active model is edited');
    AssertEquals_DINT(Expected := 7, Actual := _u.ParCfg.Speed, Message := 'live');
    AssertEquals_DINT(Expected := 7, Actual := _rec0.Speed,
        Message := 'and in its record, so a changeover back keeps it');
    _w2 := TRUE;
END_IF
TEST_FINISHED();
END_METHOD

METHOD An_unknown_model_is_refused
TEST('An_unknown_model_is_refused');
_M_Arm();
IF NOT _w3 THEN
    AssertFalse(Condition := _u.WriteModelConfig(ModelIndex := 9, TargetPath := 'Test.Model',
        WriteKey := 'probe.speed', Revision := 1, TextValue := '30'),
        Message := 'a write for a model the root does not offer is refused');
    AssertFalse(Condition := _M_Find(ModelIndex := 9, WriteKey := 'probe.speed'),
        Message := 'and so is a query');
    _w3 := TRUE;
END_IF
TEST_FINISHED();
END_METHOD

// One page, not the whole station manifest: an HMI reading another model
// must not walk every module's capabilities to find four values.
METHOD Another_model_page_holds_only_its_model_data
TEST('Another_model_page_holds_only_its_model_data');
_M_Arm();
IF NOT _w4 THEN
    AssertFalse(Condition := _M_Find(ModelIndex := 2, WriteKey := 'probe.limit'),
        Message := 'station data is not part of another model$'s page');
    AssertEquals_INT(Expected := 1, Actual := _page.EntryCount,
        Message := 'the page holds the model data and nothing else');
    AssertEquals_INT(Expected := 1, Actual := _page.PageCount,
        Message := 'so it is one page');
    AssertTrue(Condition := _M_Find(ModelIndex := 0, WriteKey := 'probe.limit'),
        Message := 'the running model$'s page is still the whole manifest');
    AssertFalse(Condition := _entry.ModelScoped,
        Message := 'where station data is marked as not model-scoped');
    _w4 := TRUE;
END_IF
TEST_FINISHED();
END_METHOD

END_FUNCTION_BLOCK

// ---- Fraktal_Tests/FB_Sha256_Tests.TcPOU
// §14 under test: F_Sha256 against the FIPS 180-4 example vectors - the empty
// message, one block, and a message whose padding spills into a second block.
FUNCTION_BLOCK FB_Sha256_Tests EXTENDS TcUnit.FB_TestSuite
VAR
    _digest : ARRAY[0..31] OF BYTE;
END_VAR

The_empty_message_hashes_to_the_published_digest();
One_block_hashes_to_the_published_digest();
Two_blocks_hash_to_the_published_digest();

// The digest of Text as 64 lowercase hex characters.
METHOD PRIVATE _M_Hex : STRING(64)
VAR_INPUT
    Text : STRING(80);
END_VAR
VAR
    i : INT;
    nib : BYTE;
    hex : STRING(16) := '0123456789abcdef';
    out : STRING(64);
    pOut : POINTER TO BYTE;
    pHex : POINTER TO BYTE;
END_VAR
F_Sha256(pData := ADR(Text), Size := INT_TO_UDINT(LEN(Text)), Digest := _digest);
pOut := ADR(out);
pHex := ADR(hex);
FOR i := 0 TO 31 DO
    nib := SHR(_digest[i], 4);
    pOut[2 * i] := pHex[nib];
    nib := _digest[i] AND 16#0F;
    pOut[2 * i + 1] := pHex[nib];
END_FOR
pOut[64] := 0;
_M_Hex := out;
END_METHOD

METHOD The_empty_message_hashes_to_the_published_digest
TEST('The_empty_message_hashes_to_the_published_digest');
AssertEquals_STRING(
    Expected := 'e3b0c44298fc1c149afbf4c8996fb92427ae41e4649b934ca495991b7852b855',
    Actual := _M_Hex(Text := ''), Message := 'SHA-256 of the empty message');
TEST_FINISHED();
END_METHOD

METHOD One_block_hashes_to_the_published_digest
TEST('One_block_hashes_to_the_published_digest');
AssertEquals_STRING(
    Expected := 'ba7816bf8f01cfea414140de5dae2223b00361a396177a9cb410ff61f20015ad',
    Actual := _M_Hex(Text := 'abc'), Message := 'SHA-256 of abc');
TEST_FINISHED();
END_METHOD

METHOD Two_blocks_hash_to_the_published_digest
TEST('Two_blocks_hash_to_the_published_digest');
AssertEquals_STRING(
    Expected := '248d6a61d20638b8e5c026930c3e6039a33ce45964ff2167f6ecedd419db06c1',
    Actual := _M_Hex(Text := 'abcdbcdecdefdefgefghfghighijhijkijkljklmklmnlmnomnopnopq'),
    Message := 'SHA-256 of the 56-byte FIPS message (padding needs a second block)');
TEST_FINISHED();
END_METHOD

END_FUNCTION_BLOCK

// ---- Fraktal_Tests/FB_AccessPersistence_Tests.TcPOU
// Core §7.7(c)/§14 under test: the hidden local user table is retained through the
// real TwinCAT file service, in the real Boot directory of the runtime.
//
// The provider keeps its default medium: a file medium in the Boot directory,
// '<key>.a' and '<key>.b' (FB_FilePersistMedium; the medium itself is covered by
// FB_PersistMedium_Tests). A "restart" here is a second provider instance over
// the same retained files - exactly what a cold start, a download or a power
// cycle leaves a new run with. Each test uses its own per-run key, so tests run
// side by side and a previous run's files or confirmation marker can never decide
// this run's result; every test removes its files when it finishes. A real
// runtime restart with the same instance (the confirmation marker) is accepted
// separately.
FUNCTION_BLOCK FB_AccessPersistence_Tests EXTENDS TcUnit.FB_TestSuite
VAR
    _tag : STRING(24);                    // per-run suffix of every key
    _garbage : ARRAY[0..15] OF BYTE := [16(16#5A)];
    _s1 : INT;
    _t1 : TON;
    _p1a : FB_LocalAccessProvider;
    _p1b : FB_LocalAccessProvider;
    _p1c : FB_LocalAccessProvider;
    _f1 : FB_ProbeFileOps;
    _s2 : INT;
    _t2 : TON;
    _p2a : FB_LocalAccessProvider;
    _p2b : FB_LocalAccessProvider;
    _f2 : FB_ProbeFileOps;
    _s3 : INT;
    _t3 : TON;
    _p3a : FB_LocalAccessProvider;
    _p3b : FB_LocalAccessProvider;
    _f3 : FB_ProbeFileOps;
    _s4 : INT;
    _t4 : TON;
    _u4a : FB_ProbeUnit;
    _u4b : FB_ProbeUnit;
    _u4c : FB_ProbeUnit;
    _p4a : FB_LocalAccessProvider;
    _p4b : FB_LocalAccessProvider;
    _p4c : FB_LocalAccessProvider;
    _f4 : FB_ProbeFileOps;
    _u5 : FB_ProbeUnit;
    _store5 : FB_ProbeAccessStore;
    _done5 : BOOL;                        // state-changing: runs exactly once
    _p6 : FB_LocalAccessProvider;
    _done6 : BOOL;                        // state-changing: runs exactly once
END_VAR
VAR CONSTANT
    TEST_TIMEOUT : TIME := T#40S;
END_VAR

IF _tag = '' THEN
    _tag := ULINT_TO_STRING(Tc2_Utilities.F_GetSystemTime() MOD 1000000000000);
END_IF
A_retained_table_survives_a_restart_and_follows_changes();
A_corrupt_table_is_announced_once_and_replaced();
A_torn_newest_image_falls_back_to_the_previous_one();
A_root_restores_logs_in_and_out_and_announces_a_lost_table();
A_root_announces_a_failed_save_and_a_lost_table_once();
Storage_names_are_bounded_and_fixed_before_restore();

METHOD PRIVATE _M_Stem : STRING(80)
VAR_INPUT
    Name : STRING(40);
END_VAR
_M_Stem := CONCAT(CONCAT('FrkTest_', Name), CONCAT('_', _tag));
END_METHOD

// The retained file of one slot, as the file medium names it ('<key>.a').
METHOD PRIVATE _M_File : STRING(255)
VAR_INPUT
    Name : STRING(40);
    SlotB : BOOL;
END_VAR
IF SlotB THEN
    _M_File := CONCAT(_M_Stem(Name := Name), '.b');
ELSE
    _M_File := CONCAT(_M_Stem(Name := Name), '.a');
END_IF
END_METHOD

METHOD PRIVATE _M_LevelOf : DINT
VAR_INPUT
    Provider : I_AccessProvider;
    User : STRING(32);
    Pin : STRING(32);
END_VAR
_M_LevelOf := TO_DINT(Provider.Authenticate(User := User, Secret := Pin));
END_METHOD

// Restart retention, a PIN change and a level change all come back from storage.
METHOD A_retained_table_survives_a_restart_and_follows_changes
TEST('A_retained_table_survives_a_restart_and_follows_changes');
_t1(IN := _s1 < 99, PT := TEST_TIMEOUT);
IF _t1.Q AND (_s1 < 99) THEN
    AssertTrue(Condition := FALSE, Message := CONCAT('timed out in step ', INT_TO_STRING(_s1)));
    _s1 := 99;
    TEST_FINISHED();
    RETURN;
END_IF
_f1.Cyclic();
CASE _s1 OF
    0:
        AssertTrue(Condition := _p1a.M_UseKey(Key := _M_Stem(Name := 'Retain')),
            Message := 'a valid key is accepted before the restore');
        // Registered BEFORE the restore finishes: kept, and written.
        _p1a.Register(User := 'op', Pin := '1234', Level := E_AccessLevel.OPERATOR);
        _p1a.Register(User := 'eng', Pin := '5678', Level := E_AccessLevel.ENGINEER);
        _s1 := 1;
    1:
        _p1a.M_Service();
        IF _p1a.Durable THEN
            AssertFalse(Condition := _p1a.M_RestoreLost(),
                Message := 'a store that never existed lost nothing');
            AssertTrue(Condition := _p1b.M_UseKey(Key := _M_Stem(Name := 'Retain')),
                Message := 'the restarted instance opens the same store');
            _s1 := 2;
        END_IF
    2:
        _p1b.M_Service();
        IF _p1b.Restored THEN
            AssertEquals_DINT(Expected := TO_DINT(E_AccessLevel.OPERATOR),
                Actual := _M_LevelOf(Provider := _p1b, User := 'op', Pin := '1234'),
                Message := 'an operator registered before the restart logs in after it');
            AssertEquals_DINT(Expected := TO_DINT(E_AccessLevel.ENGINEER),
                Actual := _M_LevelOf(Provider := _p1b, User := 'eng', Pin := '5678'),
                Message := 'every retained user keeps its level');
            AssertEquals_DINT(Expected := TO_DINT(E_AccessLevel.NONE),
                Actual := _M_LevelOf(Provider := _p1b, User := 'op', Pin := '0000'),
                Message := 'a wrong PIN is still refused after the restore');
            AssertFalse(Condition := _p1b.M_RestoreLost(), Message := 'nothing was lost');
            // Access change: a new PIN for one user, a new level for another.
            _p1b.Register(User := 'op', Pin := '2468', Level := E_AccessLevel.OPERATOR);
            _p1b.Register(User := 'eng', Pin := '5678', Level := E_AccessLevel.TECHNICIAN);
            _s1 := 3;
        END_IF
    3:
        _p1b.M_Service();
        IF _p1b.Durable THEN
            _p1c.M_UseKey(Key := _M_Stem(Name := 'Retain'));
            _s1 := 4;
        END_IF
    4:
        _p1c.M_Service();
        IF _p1c.Restored THEN
            AssertEquals_DINT(Expected := TO_DINT(E_AccessLevel.NONE),
                Actual := _M_LevelOf(Provider := _p1c, User := 'op', Pin := '1234'),
                Message := 'the replaced PIN does not come back after the next restart');
            AssertEquals_DINT(Expected := TO_DINT(E_AccessLevel.OPERATOR),
                Actual := _M_LevelOf(Provider := _p1c, User := 'op', Pin := '2468'),
                Message := 'the new PIN is the retained one');
            AssertEquals_DINT(Expected := TO_DINT(E_AccessLevel.TECHNICIAN),
                Actual := _M_LevelOf(Provider := _p1c, User := 'eng', Pin := '5678'),
                Message := 'the changed level is the retained one');
            _f1.M_Delete(Path := _M_File(Name := 'Retain', SlotB := FALSE), Where := Tc2_System.PATH_BOOTPATH);
            _s1 := 5;
        END_IF
    5:
        IF NOT _f1.Busy THEN
            _f1.M_Delete(Path := _M_File(Name := 'Retain', SlotB := TRUE), Where := Tc2_System.PATH_BOOTPATH);
            _s1 := 6;
        END_IF
    6:
        IF NOT _f1.Busy THEN
            _s1 := 99;
            TEST_FINISHED();
        END_IF
    99:
        ;
ELSE
    _s1 := 99;
END_CASE
END_METHOD

// Both slots unreadable: the loss is reported, nothing half-restored, and what
// survived is written back so the NEXT restart is silent and complete.
METHOD A_corrupt_table_is_announced_once_and_replaced
TEST('A_corrupt_table_is_announced_once_and_replaced');
_t2(IN := _s2 < 99, PT := TEST_TIMEOUT);
IF _t2.Q AND (_s2 < 99) THEN
    AssertTrue(Condition := FALSE, Message := CONCAT('timed out in step ', INT_TO_STRING(_s2)));
    _s2 := 99;
    TEST_FINISHED();
    RETURN;
END_IF
_f2.Cyclic();
CASE _s2 OF
    0:
        IF _f2.M_Write(Path := _M_File(Name := 'Corrupt', SlotB := FALSE),
            Where := Tc2_System.PATH_BOOTPATH, pData := ADR(_garbage), Size := SIZEOF(_garbage)) THEN
            _s2 := 1;
        END_IF
    1:
        IF NOT _f2.Busy AND _f2.M_Write(Path := _M_File(Name := 'Corrupt', SlotB := TRUE),
            Where := Tc2_System.PATH_BOOTPATH, pData := ADR(_garbage), Size := SIZEOF(_garbage)) THEN
            _s2 := 2;
        END_IF
    2:
        IF NOT _f2.Busy THEN
            AssertFalse(Condition := _f2.Error, Message := 'the damaged images were staged');
            _p2a.M_UseKey(Key := _M_Stem(Name := 'Corrupt'));
            _s2 := 3;
        END_IF
    3:
        _p2a.M_Service();
        IF _p2a.Restored THEN
            AssertTrue(Condition := _p2a.M_RestoreLost(),
                Message := 'two unreadable images are a loss, never a silent empty table');
            AssertEquals_DINT(Expected := TO_DINT(E_AccessLevel.NONE),
                Actual := _M_LevelOf(Provider := _p2a, User := 'op', Pin := '1234'),
                Message := 'nothing is half-restored from a corrupt image');
            _s2 := 4;
        END_IF
    4:
        _p2a.M_Service();
        IF _p2a.Durable THEN
            // Recovery is re-registration, the commissioning path a station already has.
            _p2a.Register(User := 'op', Pin := '1234', Level := E_AccessLevel.OPERATOR);
            _s2 := 5;
        END_IF
    5:
        _p2a.M_Service();
        IF _p2a.Durable THEN
            _p2b.M_UseKey(Key := _M_Stem(Name := 'Corrupt'));
            _s2 := 6;
        END_IF
    6:
        _p2b.M_Service();
        IF _p2b.Restored THEN
            AssertFalse(Condition := _p2b.M_RestoreLost(),
                Message := 'the rewritten baseline restores silently: the loss was announced once');
            AssertEquals_DINT(Expected := TO_DINT(E_AccessLevel.OPERATOR),
                Actual := _M_LevelOf(Provider := _p2b, User := 'op', Pin := '1234'),
                Message := 'the re-registered user is retained');
            _f2.M_Delete(Path := _M_File(Name := 'Corrupt', SlotB := FALSE), Where := Tc2_System.PATH_BOOTPATH);
            _s2 := 7;
        END_IF
    7:
        IF NOT _f2.Busy THEN
            _f2.M_Delete(Path := _M_File(Name := 'Corrupt', SlotB := TRUE), Where := Tc2_System.PATH_BOOTPATH);
            _s2 := 8;
        END_IF
    8:
        IF NOT _f2.Busy THEN
            _s2 := 99;
            TEST_FINISHED();
        END_IF
    99:
        ;
ELSE
    _s2 := 99;
END_CASE
END_METHOD

// A write interrupted mid-file leaves the other slot intact: the restore takes the
// newest image that validates and never mixes records from the two.
METHOD A_torn_newest_image_falls_back_to_the_previous_one
TEST('A_torn_newest_image_falls_back_to_the_previous_one');
_t3(IN := _s3 < 99, PT := TEST_TIMEOUT);
IF _t3.Q AND (_s3 < 99) THEN
    AssertTrue(Condition := FALSE, Message := CONCAT('timed out in step ', INT_TO_STRING(_s3)));
    _s3 := 99;
    TEST_FINISHED();
    RETURN;
END_IF
_f3.Cyclic();
CASE _s3 OF
    0:
        _p3a.M_UseKey(Key := _M_Stem(Name := 'Torn'));
        _p3a.Register(User := 'op', Pin := '1111', Level := E_AccessLevel.OPERATOR);
        _s3 := 1;
    1:
        _p3a.M_Service();
        IF _p3a.Durable THEN            // generation 1 in slot A
            _p3a.Register(User := 'eng', Pin := '2222', Level := E_AccessLevel.ENGINEER);
            _s3 := 2;
        END_IF
    2:
        _p3a.M_Service();
        IF _p3a.Durable THEN            // generation 2 in slot B: now tear it
            IF _f3.M_Write(Path := _M_File(Name := 'Torn', SlotB := TRUE),
                Where := Tc2_System.PATH_BOOTPATH, pData := ADR(_garbage), Size := SIZEOF(_garbage)) THEN
                _s3 := 3;
            END_IF
        END_IF
    3:
        IF NOT _f3.Busy THEN
            _p3b.M_UseKey(Key := _M_Stem(Name := 'Torn'));
            _s3 := 4;
        END_IF
    4:
        _p3b.M_Service();
        IF _p3b.Restored THEN
            AssertEquals_DINT(Expected := TO_DINT(E_AccessLevel.OPERATOR),
                Actual := _M_LevelOf(Provider := _p3b, User := 'op', Pin := '1111'),
                Message := 'the previous complete image is restored');
            AssertEquals_DINT(Expected := TO_DINT(E_AccessLevel.NONE),
                Actual := _M_LevelOf(Provider := _p3b, User := 'eng', Pin := '2222'),
                Message := 'no record of the torn image is used');
            _f3.M_Delete(Path := _M_File(Name := 'Torn', SlotB := FALSE), Where := Tc2_System.PATH_BOOTPATH);
            _s3 := 5;
        END_IF
    5:
        IF NOT _f3.Busy THEN
            _f3.M_Delete(Path := _M_File(Name := 'Torn', SlotB := TRUE), Where := Tc2_System.PATH_BOOTPATH);
            _s3 := 6;
        END_IF
    6:
        IF NOT _f3.Busy THEN
            _s3 := 99;
            TEST_FINISHED();
        END_IF
    99:
        ;
ELSE
    _s3 := 99;
END_CASE
END_METHOD

// The surface a station uses: nothing but Access.Setup. The root's access manager
// drives the store, a restored user logs in and out through the data-driven
// request, and a lost table is announced through the root's §3.8b path.
METHOD A_root_restores_logs_in_and_out_and_announces_a_lost_table
TEST('A_root_restores_logs_in_and_out_and_announces_a_lost_table');
_t4(IN := _s4 < 99, PT := TEST_TIMEOUT);
IF _t4.Q AND (_s4 < 99) THEN
    AssertTrue(Condition := FALSE, Message := CONCAT('timed out in step ', INT_TO_STRING(_s4)));
    _s4 := 99;
    TEST_FINISHED();
    RETURN;
END_IF
_f4.Cyclic();
CASE _s4 OF
    0:
        _p4a.M_UseKey(Key := _M_Stem(Name := 'Root'));
        _u4a.Setup('Test.RetainA');
        _u4a();
        _u4a.Access.Setup(Provider := _p4a, pAlarmLog := ADR(_u4a.AlarmLog));
        _p4a.Register(User := 'tech', Pin := '4711', Level := E_AccessLevel.TECHNICIAN);
        _s4 := 1;
    1:
        _u4a();                         // the root, not the test, services the store
        IF _p4a.Durable THEN
            _p4b.M_UseKey(Key := _M_Stem(Name := 'Root'));
            _u4b.Setup('Test.RetainB');
            _u4b();
            _u4b.Access.Setup(Provider := _p4b, pAlarmLog := ADR(_u4b.AlarmLog));
            _s4 := 2;
        END_IF
    2:
        _u4b();
        IF _p4b.Restored THEN
            _u4b.Access.RequestLogin(User := 'tech', Secret := '4711');
            _u4b();
            AssertEquals_DINT(Expected := TO_DINT(E_AccessLevel.TECHNICIAN),
                Actual := TO_DINT(_u4b.Access.CurrentLevel),
                Message := 'a user retained by another run logs in through the root');
            _u4b.Access.RequestLogout();
            _u4b();
            AssertEquals_DINT(Expected := TO_DINT(E_AccessLevel.NONE),
                Actual := TO_DINT(_u4b.Access.CurrentLevel), Message := 'and logs out');
            _u4b.Access.RequestLogin(User := 'tech', Secret := '0000');
            _u4b();
            AssertTrue(Condition := _u4b.Access.LoginFailed,
                Message := 'a wrong PIN for a retained user is refused');
            AssertFalse(Condition := _u4b.ConfigPersist.RestoreLost,
                Message := 'a good table is not a loss');
            _s4 := 3;
        END_IF
    3:
        IF _f4.M_Write(Path := _M_File(Name := 'Root', SlotB := FALSE),
            Where := Tc2_System.PATH_BOOTPATH, pData := ADR(_garbage), Size := SIZEOF(_garbage)) THEN
            _s4 := 4;
        END_IF
    4:
        IF NOT _f4.Busy AND _f4.M_Write(Path := _M_File(Name := 'Root', SlotB := TRUE),
            Where := Tc2_System.PATH_BOOTPATH, pData := ADR(_garbage), Size := SIZEOF(_garbage)) THEN
            _s4 := 5;
        END_IF
    5:
        IF NOT _f4.Busy THEN
            _p4c.M_UseKey(Key := _M_Stem(Name := 'Root'));
            _u4c.Setup('Test.RetainC');
            _u4c();
            _u4c.Access.Setup(Provider := _p4c, pAlarmLog := ADR(_u4c.AlarmLog));
            _s4 := 6;
        END_IF
    6:
        _u4c();
        IF _p4c.Restored THEN
            _u4c();                     // the root drains the loss on its next scan
            _u4c();
            AssertTrue(Condition := _u4c.ConfigPersist.RestoreLost,
                Message := 'a lost user table is published like any lost image (3.8b)');
            AssertEquals_STRING(Expected := 'Test.RetainC.Access',
                Actual := _u4c.ConfigPersist.LostPath, Message := 'naming the access table');
            AssertTrue(Condition := F_ProbeAlarmActive(pLog := ADR(_u4c.AlarmLog),
                Reason := E_Reason.CONFIG_RESTORE_LOST, Source := 'Test.RetainC.Access'),
                Message := 'and announced until an engineer acknowledges it');
            _u4c.Access.RequestLogin(User := 'tech', Secret := '4711');
            _u4c();
            AssertEquals_DINT(Expected := TO_DINT(E_AccessLevel.NONE),
                Actual := TO_DINT(_u4c.Access.CurrentLevel),
                Message := 'a user from a lost table cannot log in');
            _s4 := 7;
        END_IF
    7:
        _u4c();
        IF _p4c.Durable AND _f4.M_Delete(Path := _M_File(Name := 'Root', SlotB := FALSE),
            Where := Tc2_System.PATH_BOOTPATH) THEN
            _s4 := 8;
        END_IF
    8:
        IF NOT _f4.Busy THEN
            _f4.M_Delete(Path := _M_File(Name := 'Root', SlotB := TRUE), Where := Tc2_System.PATH_BOOTPATH);
            _s4 := 9;
        END_IF
    9:
        IF NOT _f4.Busy THEN
            _s4 := 99;
            TEST_FINISHED();
        END_IF
    99:
        ;
ELSE
    _s4 := 99;
END_CASE
END_METHOD

// The root's side of a retained table, with the store's outcomes forced: a write
// that cannot be made durable is CONFIG_PERSIST_FAILED until a later one succeeds,
// and a lost table reaches the root's §3.8b restore annunciation exactly once.
// (The provider's own failing write is accepted live, against a real Boot folder.)
METHOD A_root_announces_a_failed_save_and_a_lost_table_once
TEST('A_root_announces_a_failed_save_and_a_lost_table_once');
IF _done5 THEN
    RETURN;
END_IF
_done5 := TRUE;
_u5.Setup('Test.StoreRoot');
_u5();
_u5.Access.Setup(Provider := _store5, pAlarmLog := ADR(_u5.AlarmLog));
_u5();
AssertTrue(Condition := _store5.Serviced > 0,
    Message := 'the root services a provider that retains its table: the project calls nothing');
_store5.SaveFailed := TRUE;
_u5();
AssertTrue(Condition := F_ProbeAlarmActive(pLog := ADR(_u5.AlarmLog),
    Reason := E_Reason.CONFIG_PERSIST_FAILED, Source := 'Access'),
    Message := 'a registration that cannot be written is announced, not swallowed');
AssertFalse(Condition := _u5.AlarmLog.Blocking,
    Message := 'it does not stop a machine that can still finish its parts');
_store5.SaveFailed := FALSE;
_u5();
AssertFalse(Condition := F_ProbeAlarmActive(pLog := ADR(_u5.AlarmLog),
    Reason := E_Reason.CONFIG_PERSIST_FAILED, Source := 'Access'),
    Message := 'a later successful write clears the announcement');
_store5.RestoreLost := TRUE;
_u5();
_u5();
AssertTrue(Condition := _u5.ConfigPersist.RestoreLost,
    Message := 'a lost table is published by the root (3.8b)');
AssertEquals_STRING(Expected := 'Test.StoreRoot.Access', Actual := _u5.ConfigPersist.LostPath,
    Message := 'naming the access table');
AssertTrue(Condition := F_ProbeAlarmActive(pLog := ADR(_u5.AlarmLog),
    Reason := E_Reason.CONFIG_RESTORE_LOST, Source := 'Test.StoreRoot.Access'),
    Message := 'and annunciated with that path');
AssertFalse(Condition := _u5.Access.M_TakeRestoreLoss(),
    Message := 'the root took it once: a standing loss is not re-announced every scan');
TEST_FINISHED();
END_METHOD

METHOD Storage_names_are_bounded_and_fixed_before_restore
TEST('Storage_names_are_bounded_and_fixed_before_restore');
IF _done6 THEN
    RETURN;
END_IF
_done6 := TRUE;
AssertFalse(Condition := _p6.M_UseKey(Key := '..\Boot'),
    Message := 'a path separator can never leave the medium$'s folder');
AssertFalse(Condition := _p6.M_UseKey(Key := 'two words'),
    Message := 'only letters, digits, underscore, dot and dash are accepted');
AssertTrue(Condition := _p6.M_UseKey(Key := ''),
    Message := 'an empty key keeps the table volatile by choice');
_p6.M_Service();
AssertTrue(Condition := _p6.Restored, Message := 'a volatile table is restored at once');
AssertFalse(Condition := _p6.Durable, Message := 'and never claims durability');
AssertFalse(Condition := _p6.M_UseKey(Key := 'Later'),
    Message := 'a started store cannot be retargeted');
AssertFalse(Condition := _p6.Register(User := '', Pin := '1', Level := E_AccessLevel.OPERATOR),
    Message := 'an unnamed user is refused');
AssertTrue(Condition := _p6.Register(User := 'op', Pin := '1', Level := E_AccessLevel.OPERATOR),
    Message := 'a named user is accepted');
TEST_FINISHED();
END_METHOD

END_FUNCTION_BLOCK

// ---- Fraktal_Tests/FB_ProbeAccessStore.TcPOU
// Test double: an access provider that also retains its table, with every store
// outcome settable, so a root's handling of a failed save or a lost table is
// tested without staging damage on the runtime's file system.
FUNCTION_BLOCK FB_ProbeAccessStore IMPLEMENTS I_AccessProvider, I_AccessStore
VAR_INPUT
    RestoreLost : BOOL;
    SaveFailed  : BOOL;
END_VAR
VAR_OUTPUT
    Serviced : UDINT;           // M_Service calls received
END_VAR

;

METHOD Authenticate : E_AccessLevel
VAR_INPUT
    User : STRING(32);
    Secret : STRING(32);
END_VAR
Authenticate := E_AccessLevel.NONE;
END_METHOD

METHOD M_Service : BOOL
Serviced := Serviced + 1;
M_Service := TRUE;
END_METHOD

METHOD M_RestoreLost : BOOL
M_RestoreLost := RestoreLost;
END_METHOD

METHOD M_SaveFailed : BOOL
M_SaveFailed := SaveFailed;
END_METHOD

END_FUNCTION_BLOCK

// ---- Fraktal_Tests/F_ProbeAlarmActive.TcPOU
// Test helper: is an event with this reason and source currently active in Log?
FUNCTION F_ProbeAlarmActive : BOOL
VAR_INPUT
    pLog   : POINTER TO FB_AlarmLog;
    Reason : E_Reason;
    Source : STRING(255);
END_VAR
VAR
    i : INT;
END_VAR

F_ProbeAlarmActive := FALSE;
IF pLog = 0 THEN
    RETURN;
END_IF
FOR i := 1 TO MIN(pLog^.NActive, PL_Fraktal.MAX_ALARM_ACTIVE) DO
    IF (pLog^.Active[i].ReasonCode = Reason) AND (pLog^.Active[i].SourcePath = Source) THEN
        F_ProbeAlarmActive := TRUE;
    END_IF
END_FOR

END_FUNCTION

// ---- Fraktal_Tests/FB_PlatformHealth_Tests.TcPOU
// TC3 §8.12/§10.5 under test: what the target-specific providers publish when a
// metric is measured, stale, out of range or not offered by the hardware. The
// providers' measurement seams (M_ApplyReading, M_ApplyMasterSample) are the same
// calls their own ADS state machines make, so these are the real evaluations.
FUNCTION_BLOCK FB_PlatformHealth_Tests EXTENDS TcUnit.FB_TestSuite
VAR
    _log : FB_AlarmLog;
    _health : FB_SystemHealthPublisher;
    _input : ST_SystemHealthInput;
    _fresh : ST_SystemHealthInput;
    _cfg : ST_SystemHealthParCfg;
    _ipc : FB_TcIpcDiagnostics;
    _bus : FB_EcBusHealth;
    _values : ARRAY[1..8] OF LREAL;
    _done : ARRAY[1..3] OF BOOL;
END_VAR

Unmeasured_fan_and_storage_raise_nothing();
Ipc_metrics_are_available_only_while_measured();
EtherCat_master_counts_windows_and_dc();

// Core §8.12 "where the hardware exposes them": a fanless IPC or a drive without
// wear data is not a fault, and not a healthy reading either.
METHOD Unmeasured_fan_and_storage_raise_nothing
TEST('Unmeasured_fan_and_storage_raise_nothing');
IF _done[1] THEN
    RETURN;
END_IF
_done[1] := TRUE;
AssertTrue(Condition := _fresh.FanAvailable AND _fresh.StorageAvailable,
    Message := 'a producer that never sets the new flags keeps the single IPC meaning');
_health.Setup(SourcePath := 'Test.Platform.SystemHealth', pAlarmLog := ADR(_log));
_input.TaskAvailable := TRUE;
_input.TaskCycleUs := 1000;
_input.ControllerAvailable := TRUE;
_input.CpuLoadPct := 10.0;
_input.MemoryAvailableMb := 1024;
_input.IpcAvailable := TRUE;
_input.IpcTemperatureC := 40.0;
_input.FanAvailable := FALSE;
_input.FanHealthy := FALSE;
_input.StorageAvailable := FALSE;
_input.StorageHealthPct := 0.0;
_input.TimeQuality.Available := TRUE;
_input.TimeQuality.Synchronized := TRUE;
_health.Cyclic(Input := _input, ParCfg := _cfg, Configured := TRUE);
AssertFalse(Condition := F_ProbeAlarmActive(pLog := ADR(_log), Reason := E_Reason.IPC_FAN_FAULT,
    Source := 'Test.Platform.SystemHealth'), Message := 'no fan to measure is no fan fault');
AssertFalse(Condition := F_ProbeAlarmActive(pLog := ADR(_log), Reason := E_Reason.STORAGE_HEALTH_LOW,
    Source := 'Test.Platform.SystemHealth'), Message := 'no wear data is no storage fault');
AssertFalse(Condition := _health.Status.FanAvailable OR _health.Status.StorageAvailable,
    Message := 'the published status says the readings are not measurements');
_input.FanAvailable := TRUE;
_input.StorageAvailable := TRUE;
_health.Cyclic(Input := _input, ParCfg := _cfg, Configured := TRUE);
AssertTrue(Condition := F_ProbeAlarmActive(pLog := ADR(_log), Reason := E_Reason.IPC_FAN_FAULT,
    Source := 'Test.Platform.SystemHealth'), Message := 'a measured stopped fan is a fault');
AssertTrue(Condition := F_ProbeAlarmActive(pLog := ADR(_log), Reason := E_Reason.STORAGE_HEALTH_LOW,
    Source := 'Test.Platform.SystemHealth'), Message := 'measured worn storage is a fault');
_input.FanHealthy := TRUE;
_input.StorageHealthPct := 90.0;
_health.Cyclic(Input := _input, ParCfg := _cfg, Configured := TRUE);
AssertFalse(Condition := F_ProbeAlarmActive(pLog := ADR(_log), Reason := E_Reason.IPC_FAN_FAULT,
    Source := 'Test.Platform.SystemHealth'), Message := 'a turning fan clears it');
AssertFalse(Condition := F_ProbeAlarmActive(pLog := ADR(_log), Reason := E_Reason.STORAGE_HEALTH_LOW,
    Source := 'Test.Platform.SystemHealth'), Message := 'healthy storage clears it');
TEST_FINISHED();
END_METHOD

METHOD Ipc_metrics_are_available_only_while_measured
TEST('Ipc_metrics_are_available_only_while_measured');
IF _done[2] THEN
    RETURN;
END_IF
_done[2] := TRUE;
AssertFalse(Condition := _ipc.ControllerAvailable OR _ipc.IpcAvailable
    OR _ipc.FanAvailable OR _ipc.StorageAvailable,
    Message := 'nothing is available before it was measured');
_values[1] := 35.0;
AssertTrue(Condition := _ipc.M_ApplyReading(Metric := 0, Ok := TRUE, Values := _values,
    Count := 1, MonoNow := T#10S), Message := 'CPU usage accepted');
AssertFalse(Condition := _ipc.ControllerAvailable,
    Message := 'controller metrics need CPU AND memory');
_values[1] := 2147483648.0;     // 2 GiB available program memory
_ipc.M_ApplyReading(Metric := 1, Ok := TRUE, Values := _values, Count := 1, MonoNow := T#12S);
AssertTrue(Condition := _ipc.ControllerAvailable, Message := 'both measured: available');
AssertEquals_LREAL(Expected := 35.0, Actual := _ipc.CpuLoadPct, Delta := 0.001,
    Message := 'CPU usage in percent');
AssertEquals_UDINT(Expected := 2048, Actual := _ipc.MemoryAvailableMb,
    Message := 'available program memory in MB');
_values[1] := 120.0;
AssertFalse(Condition := _ipc.M_ApplyReading(Metric := 0, Ok := TRUE, Values := _values,
    Count := 1, MonoNow := T#14S), Message := 'an impossible CPU reading is refused');
AssertEquals_LREAL(Expected := 35.0, Actual := _ipc.CpuLoadPct, Delta := 0.001,
    Message := 'and does not replace the last measurement');
AssertFalse(Condition := _ipc.M_ApplyReading(Metric := 0, Ok := FALSE, Values := _values,
    Count := 0, MonoNow := T#30S), Message := 'a failed read is reported');
_values[1] := 55.0;
_values[2] := 61.0;
_ipc.M_ApplyReading(Metric := 2, Ok := TRUE, Values := _values, Count := 2, MonoNow := T#55S);
AssertTrue(Condition := _ipc.IpcAvailable, Message := 'temperature measured');
AssertEquals_LREAL(Expected := 61.0, Actual := _ipc.IpcTemperatureC, Delta := 0.001,
    Message := 'the hottest CPU reading is the IPC temperature');
AssertFalse(Condition := _ipc.ControllerAvailable,
    Message := 'no fresh CPU or memory reading for over 40 s: controller metrics expire');
_values[1] := 1800.0;
_values[2] := 0.0;
_ipc.M_ApplyReading(Metric := 3, Ok := TRUE, Values := _values, Count := 2, MonoNow := T#56S);
AssertTrue(Condition := _ipc.FanAvailable AND NOT _ipc.FanHealthy,
    Message := 'one stopped fan of two is a measured fan fault');
_values[1] := 80.0;
_values[2] := 60.0;
_ipc.M_ApplyReading(Metric := 4, Ok := TRUE, Values := _values, Count := 2, MonoNow := T#57S);
AssertFalse(Condition := _ipc.StorageAvailable,
    Message := 'storage health needs both wear figures');
_values[1] := 90.0;
_ipc.M_ApplyReading(Metric := 5, Ok := TRUE, Values := _values, Count := 1, MonoNow := T#58S);
AssertTrue(Condition := _ipc.StorageAvailable, Message := 'both wear figures measured');
AssertEquals_LREAL(Expected := 60.0, Actual := _ipc.StorageHealthPct, Delta := 0.001,
    Message := 'the worst figure of the worst drive');
AssertFalse(Condition := _ipc.M_ApplyReading(Metric := 6, Ok := TRUE, Values := _values,
    Count := 1, MonoNow := T#59S), Message := 'an unknown metric is refused');
TEST_FINISHED();
END_METHOD

// The master's counters are cumulative since it started. Losses during start-up
// must not count, a burst must be held long enough to be seen, a cleared counter
// must not underflow, and DC and the slave states are read from the device state.
METHOD EtherCat_master_counts_windows_and_dc
TEST('EtherCat_master_counts_windows_and_dc');
IF _done[3] THEN
    RETURN;
END_IF
_done[3] := TRUE;
AssertFalse(Condition := _bus.MasterAvailable OR _bus.MasterHealthy OR _bus.DcSynchronized,
    Message := 'an unread master is neither available nor healthy');
_bus.M_ApplyMasterSample(Ok := TRUE, DevState := 0, LostFrames := 100, CrcErrors := 5,
    MonoNow := T#1S);
AssertTrue(Condition := _bus.MasterAvailable AND _bus.MasterHealthy AND _bus.DcSynchronized,
    Message := 'a clean device state is a healthy, synchronized master');
AssertEquals_UDINT(Expected := 0, Actual := _bus.LostFrameCount,
    Message := 'frames lost before the first sample are not counted');
_bus.M_ApplyMasterSample(Ok := TRUE, DevState := 0, LostFrames := 103, CrcErrors := 7,
    MonoNow := T#2S);
AssertEquals_UDINT(Expected := 3, Actual := _bus.LostFrameCount,
    Message := 'lost frames of the current window are visible at once');
AssertEquals_UDINT(Expected := 2, Actual := _bus.SlaveErrorCount,
    Message := 'and so are new CRC errors');
_bus.M_ApplyMasterSample(Ok := TRUE, DevState := 0, LostFrames := 104, CrcErrors := 7,
    MonoNow := T#12S);
_bus.M_ApplyMasterSample(Ok := TRUE, DevState := 0, LostFrames := 104, CrcErrors := 7,
    MonoNow := T#13S);
AssertEquals_UDINT(Expected := 4, Actual := _bus.LostFrameCount,
    Message := 'a burst is held for the whole next window');
_bus.M_ApplyMasterSample(Ok := TRUE, DevState := 0, LostFrames := 104, CrcErrors := 7,
    MonoNow := T#23S);
_bus.M_ApplyMasterSample(Ok := TRUE, DevState := 0, LostFrames := 104, CrcErrors := 7,
    MonoNow := T#24S);
AssertEquals_UDINT(Expected := 0, Actual := _bus.LostFrameCount,
    Message := 'a clean window clears it');
_bus.M_ApplyMasterSample(Ok := TRUE, DevState := 0, LostFrames := 2, CrcErrors := 0,
    MonoNow := T#25S);
AssertEquals_UDINT(Expected := 2, Actual := _bus.LostFrameCount,
    Message := 'a cleared counter counts from zero instead of underflowing');
_bus.M_ApplyMasterSample(Ok := TRUE, DevState := WORD#16#1000, LostFrames := 2, CrcErrors := 0,
    MonoNow := T#26S);
AssertTrue(Condition := _bus.MasterHealthy AND NOT _bus.DcSynchronized,
    Message := 'DC out of sync is reported apart from the master health');
_bus.M_ApplyMasterSample(Ok := TRUE, DevState := WORD#16#0004, LostFrames := 2, CrcErrors := 0,
    MonoNow := T#27S);
AssertTrue(Condition := _bus.MasterHealthy,
    Message := 'a redundancy-adapter link note is not a fault of the working line');
_bus.M_ApplyMasterSample(Ok := TRUE, DevState := WORD#16#0400, LostFrames := 2, CrcErrors := 0,
    MonoNow := T#28S);
AssertFalse(Condition := _bus.MasterHealthy, Message := 'a slave in SAFE-OP is not a healthy bus');
_bus.M_ApplyMasterSample(Ok := FALSE, DevState := 0, LostFrames := 0, CrcErrors := 0,
    MonoNow := T#32S);
AssertFalse(Condition := _bus.MasterAvailable OR _bus.MasterHealthy OR _bus.DcSynchronized,
    Message := 'no successful sample for more than 3 s: the master is unavailable');
AssertFalse(Condition := _bus.M_BusOk(), Message := 'and the bus is never reported valid');
TEST_FINISHED();
END_METHOD

END_FUNCTION_BLOCK

// ---- Fraktal_Tests/FB_PersistMedium_Tests.TcPOU
// Core §3.8b under test: the plug-and-play persistence media through the real
// TwinCAT file service and the real persistent-data writer of the test runtime.
// A file medium keeps the newest whole copy through a torn write, refuses a
// damaged one, reports a document it confirmed and then lost, and creates its
// folder; the retentive medium keeps a bounded pool and says when it is full.
// Every test uses per-run keys and removes what it wrote.
FUNCTION_BLOCK FB_PersistMedium_Tests EXTENDS TcUnit.FB_TestSuite
VAR
    _tag     : STRING(24);
    _docA    : ARRAY[0..99] OF BYTE;
    _docB    : ARRAY[0..199] OF BYTE;
    _buf     : ARRAY[0..299] OF BYTE;
    _small   : ARRAY[0..9] OF BYTE;
    _garbage : ARRAY[0..15] OF BYTE := [16(16#5A)];
    _filled  : BOOL;
    _s1 : INT;
    _t1 : TON;
    _k1 : UDINT;
    _r1 : ST_PersistResult;
    _m1 : FB_FilePersistMedium;
    _f1 : FB_ProbeFileOps;
    _done2 : BOOL;
    _m2 : FB_FilePersistMedium;
    _p2a : FB_LocalAccessProvider;
    _p2b : FB_LocalAccessProvider;
    _ret : FB_RetainPersistMedium;        // one pool for the whole suite (persistent)
    _s3 : INT;
    _t3 : TON;
    _k3 : UDINT;
    _r3 : ST_PersistResult;
    _n3 : INT;
    _full3 : INT;
    _s4 : INT;
    _t4 : TON;
    _k4 : UDINT;
    _r4 : ST_PersistResult;
    _m4 : FB_FilePersistMedium;
    _f4 : FB_ProbeFileOps;
    _s5 : INT;
    _t5 : TON;
    _k5 : UDINT;
    _r5 : ST_PersistResult;
    _m5 : FB_FilePersistMedium;
    _m6 : FB_FilePersistMedium;
    _m7 : FB_FilePersistMedium;
    _f5 : FB_ProbeFileOps;
END_VAR
VAR CONSTANT
    TEST_TIMEOUT : TIME := T#60S;
    GENERIC_FOLDER : STRING(80) := 'C:\ProgramData\Fraktal\Tests\Medium\';
END_VAR

IF _tag = '' THEN
    _tag := ULINT_TO_STRING(Tc2_Utilities.F_GetSystemTime() MOD 1000000000000);
END_IF
IF NOT _filled THEN
    _filled := TRUE;
    MEMSET(destAddr := ADR(_docA), fillByte := 16#41, n := SIZEOF(_docA));
    MEMSET(destAddr := ADR(_docB), fillByte := 16#42, n := SIZEOF(_docB));
    _docB[0] := 10;                     // a line break inside a document is just a byte
END_IF
A_file_document_survives_a_torn_write_and_reports_a_loss();
Requests_are_refused_or_answered_never_left_waiting();
The_retentive_pool_keeps_documents_and_says_when_it_is_full();
A_file_medium_creates_its_folder();
The_newest_copy_wins_in_either_slot();

METHOD PRIVATE _M_Key : STRING(80)
VAR_INPUT
    Name : STRING(40);
END_VAR
_M_Key := CONCAT(CONCAT('FrkMed_', Name), CONCAT('_', _tag));
END_METHOD

METHOD A_file_document_survives_a_torn_write_and_reports_a_loss
VAR
    key : STRING(80);
END_VAR
TEST('A_file_document_survives_a_torn_write_and_reports_a_loss');
_t1(IN := _s1 < 99, PT := TEST_TIMEOUT);
IF _t1.Q AND (_s1 < 99) THEN
    AssertTrue(Condition := FALSE, Message := CONCAT('timed out in step ', INT_TO_STRING(_s1)));
    _s1 := 99;
    TEST_FINISHED();
    RETURN;
END_IF
key := _M_Key(Name := 'Doc');
_f1.Cyclic();
CASE _s1 OF
    0:
        _m1.Setup(Folder := '', Where := Tc2_System.PATH_BOOTPATH);
        _k1 := _m1.M_StartWrite(Key := key, pData := ADR(_docA), Size := SIZEOF(_docA));
        AssertTrue(Condition := _k1 <> 0, Message := 'a write is queued');
        _s1 := 1;
    1:
        IF _m1.M_Poll(Ticket := _k1, Result := _r1) THEN
            AssertTrue(Condition := _r1.Ok, Message := 'the first copy is durable');
            _k1 := _m1.M_StartWrite(Key := key, pData := ADR(_docB), Size := SIZEOF(_docB));
            _s1 := 2;
        END_IF
    2:
        IF _m1.M_Poll(Ticket := _k1, Result := _r1) THEN
            AssertTrue(Condition := _r1.Ok, Message := 'the second copy is durable');
            MEMSET(destAddr := ADR(_buf), fillByte := 0, n := SIZEOF(_buf));
            _k1 := _m1.M_StartRead(Key := key, pData := ADR(_buf), Size := SIZEOF(_buf));
            _s1 := 3;
        END_IF
    3:
        IF _m1.M_Poll(Ticket := _k1, Result := _r1) THEN
            AssertTrue(Condition := _r1.Ok AND _r1.Found, Message := 'the document is read back');
            AssertFalse(Condition := _r1.Lost, Message := 'nothing was lost');
            AssertEquals_UDINT(Expected := SIZEOF(_docB), Actual := _r1.Length,
                Message := 'the newest copy, whole');
            AssertEquals_DINT(Expected := 0, Actual := MEMCMP(pBuf1 := ADR(_buf),
                pBuf2 := ADR(_docB), n := SIZEOF(_docB)), Message := 'byte for byte');
            // The second write went to slot b: tear it.
            _f1.M_Write(Path := CONCAT(key, '.b'), Where := Tc2_System.PATH_BOOTPATH,
                pData := ADR(_garbage), Size := SIZEOF(_garbage));
            _s1 := 4;
        END_IF
    4:
        IF NOT _f1.Busy THEN
            _k1 := _m1.M_StartRead(Key := key, pData := ADR(_buf), Size := SIZEOF(_buf));
            _s1 := 5;
        END_IF
    5:
        IF _m1.M_Poll(Ticket := _k1, Result := _r1) THEN
            AssertTrue(Condition := _r1.Found, Message := 'the previous whole copy is returned');
            AssertEquals_UDINT(Expected := SIZEOF(_docA), Actual := _r1.Length,
                Message := 'never a mix of the two');
            AssertEquals_DINT(Expected := 0, Actual := MEMCMP(pBuf1 := ADR(_buf),
                pBuf2 := ADR(_docA), n := SIZEOF(_docA)), Message := 'the first document');
            AssertTrue(Condition := _r1.Lost,
                Message := 'and it is older than the copy confirmed written: a loss');
            _f1.M_Write(Path := CONCAT(key, '.a'), Where := Tc2_System.PATH_BOOTPATH,
                pData := ADR(_garbage), Size := SIZEOF(_garbage));
            _s1 := 6;
        END_IF
    6:
        IF NOT _f1.Busy THEN
            _k1 := _m1.M_StartRead(Key := key, pData := ADR(_buf), Size := SIZEOF(_buf));
            _s1 := 7;
        END_IF
    7:
        IF _m1.M_Poll(Ticket := _k1, Result := _r1) THEN
            AssertTrue(Condition := _r1.Ok, Message := 'two damaged copies still get an answer');
            AssertFalse(Condition := _r1.Found, Message := 'nothing damaged is returned');
            AssertTrue(Condition := _r1.Lost, Message := 'and it is a loss');
            _f1.M_Delete(Path := CONCAT(key, '.a'), Where := Tc2_System.PATH_BOOTPATH);
            _s1 := 8;
        END_IF
    8:
        IF NOT _f1.Busy THEN
            _f1.M_Delete(Path := CONCAT(key, '.b'), Where := Tc2_System.PATH_BOOTPATH);
            _s1 := 9;
        END_IF
    9:
        IF NOT _f1.Busy THEN
            _k1 := _m1.M_StartRead(Key := key, pData := ADR(_buf), Size := SIZEOF(_buf));
            _s1 := 10;
        END_IF
    10:
        IF _m1.M_Poll(Ticket := _k1, Result := _r1) THEN
            AssertFalse(Condition := _r1.Found, Message := 'deleted files return nothing');
            AssertTrue(Condition := _r1.Lost,
                Message := 'and the persistent confirmation alone tells that from a first start');
            _k1 := _m1.M_StartWrite(Key := key, pData := ADR(_docA), Size := 0);
            _s1 := 11;
        END_IF
    11:
        IF _m1.M_Poll(Ticket := _k1, Result := _r1) THEN
            AssertTrue(Condition := _r1.Ok, Message := 'an empty document is a durable deletion');
            _k1 := _m1.M_StartRead(Key := key, pData := ADR(_buf), Size := SIZEOF(_buf));
            _s1 := 12;
        END_IF
    12:
        IF _m1.M_Poll(Ticket := _k1, Result := _r1) THEN
            AssertTrue(Condition := _r1.Ok AND NOT _r1.Found,
                Message := 'a deleted document is not there');
            AssertFalse(Condition := _r1.Lost, Message := 'by intent, so nothing was lost');
            _k1 := _m1.M_StartWrite(Key := key, pData := ADR(_docB), Size := SIZEOF(_docB));
            _s1 := 13;
        END_IF
    13:
        IF _m1.M_Poll(Ticket := _k1, Result := _r1) THEN
            _k1 := _m1.M_StartRead(Key := key, pData := ADR(_small), Size := SIZEOF(_small));
            _s1 := 14;
        END_IF
    14:
        IF _m1.M_Poll(Ticket := _k1, Result := _r1) THEN
            AssertFalse(Condition := _r1.Ok OR _r1.Found,
                Message := 'a document larger than the buffer is refused, not cut');
            AssertEquals_UDINT(Expected := 16#705, Actual := _r1.ErrorId,
                Message := 'with the size error');
            _k1 := _m1.M_StartRead(Key := _M_Key(Name := 'Never'), pData := ADR(_buf),
                Size := SIZEOF(_buf));
            _s1 := 15;
        END_IF
    15:
        IF _m1.M_Poll(Ticket := _k1, Result := _r1) THEN
            AssertTrue(Condition := _r1.Ok AND NOT _r1.Found AND NOT _r1.Lost,
                Message := 'a key never written is a first start, not a loss');
            _f1.M_Delete(Path := CONCAT(key, '.a'), Where := Tc2_System.PATH_BOOTPATH);
            _s1 := 16;
        END_IF
    16:
        IF NOT _f1.Busy THEN
            _f1.M_Delete(Path := CONCAT(key, '.b'), Where := Tc2_System.PATH_BOOTPATH);
            _s1 := 17;
        END_IF
    17:
        IF NOT _f1.Busy THEN
            _s1 := 99;
            TEST_FINISHED();
        END_IF
    99:
        ;
ELSE
    _s1 := 99;
END_CASE
END_METHOD

METHOD Requests_are_refused_or_answered_never_left_waiting
VAR
    answer : ST_PersistResult;
    queued : INT;
    i : INT;
END_VAR
TEST('Requests_are_refused_or_answered_never_left_waiting');
IF _done2 THEN
    RETURN;
END_IF
_done2 := TRUE;
AssertTrue(Condition := _m2.Setup(Folder := '', Where := Tc2_System.PATH_BOOTPATH),
    Message := 'a medium is set up before its first request');
AssertEquals_UDINT(Expected := 0, Actual := _m2.M_StartWrite(Key := 'two words',
    pData := ADR(_docA), Size := SIZEOF(_docA)), Message := 'a key with a space is refused');
AssertEquals_UDINT(Expected := 0, Actual := _m2.M_StartWrite(Key := '..\x',
    pData := ADR(_docA), Size := SIZEOF(_docA)), Message := 'a key can never leave the folder');
AssertEquals_UDINT(Expected := 0, Actual := _m2.M_StartRead(Key := '',
    pData := ADR(_buf), Size := SIZEOF(_buf)), Message := 'an empty key is refused');
AssertEquals_UDINT(Expected := 0, Actual := _m2.M_StartWrite(Key := 'k',
    pData := ADR(_docA), Size := PL_Fraktal.MAX_PERSIST_DOC_BYTES + 1),
    Message := 'a document over the bound is refused');
AssertEquals_UDINT(Expected := 0, Actual := _m2.M_StartRead(Key := 'k',
    pData := ADR(_buf), Size := 0), Message := 'a read needs a buffer');
AssertTrue(Condition := _m2.M_Poll(Ticket := 424242, Result := answer),
    Message := 'an unknown ticket finishes at once');
AssertFalse(Condition := answer.Ok, Message := 'and is not a success');
AssertEquals_UDINT(Expected := 16#706, Actual := answer.ErrorId, Message := 'it is an invalid request');
queued := 0;
FOR i := 1 TO PL_Fraktal.MAX_PERSIST_QUEUE + 1 DO
    IF _m2.M_StartRead(Key := _M_Key(Name := 'Queue'), pData := ADR(_buf),
            Size := SIZEOF(_buf)) <> 0 THEN
        queued := queued + 1;
    END_IF
END_FOR
AssertEquals_INT(Expected := PL_Fraktal.MAX_PERSIST_QUEUE, Actual := queued,
    Message := 'the queue is bounded; one more is refused, to be asked again');
AssertFalse(Condition := _m2.Setup(Folder := 'Elsewhere', Where := Tc2_System.PATH_BOOTPATH),
    Message := 'a medium in use is never retargeted');
AssertTrue(Condition := _m2.M_Confidential(), Message := 'files are not symbol-readable');
AssertEquals_DINT(Expected := TO_DINT(E_ConfigStore.FILE_JSON), Actual := TO_DINT(_m2.M_Kind()),
    Message := 'a file medium is FILE_JSON');
AssertFalse(Condition := _ret.M_Confidential(), Message := 'a persistent pool is symbol-readable');
AssertEquals_DINT(Expected := TO_DINT(E_ConfigStore.LOCAL_RETAIN), Actual := TO_DINT(_ret.M_Kind()),
    Message := 'and is LOCAL_RETAIN');
AssertFalse(Condition := _p2a.M_UseMedium(Medium := _ret),
    Message := 'a user table never goes to a symbol-readable medium (14)');
AssertTrue(Condition := _p2b.M_UseMedium(Medium := _m2),
    Message := 'a confidential medium is accepted');
TEST_FINISHED();
END_METHOD

METHOD The_retentive_pool_keeps_documents_and_says_when_it_is_full
TEST('The_retentive_pool_keeps_documents_and_says_when_it_is_full');
_t3(IN := _s3 < 99, PT := TEST_TIMEOUT);
IF _t3.Q AND (_s3 < 99) THEN
    AssertTrue(Condition := FALSE, Message := CONCAT('timed out in step ', INT_TO_STRING(_s3)));
    _s3 := 99;
    TEST_FINISHED();
    RETURN;
END_IF
CASE _s3 OF
    0:
        _k3 := _ret.M_StartWrite(Key := _M_Key(Name := 'Pool'), pData := ADR(_docB),
            Size := SIZEOF(_docB));
        _s3 := 1;
    1:
        IF _ret.M_Poll(Ticket := _k3, Result := _r3) THEN
            AssertTrue(Condition := _r3.Ok, Message := 'the document reaches the persistent image');
            MEMSET(destAddr := ADR(_buf), fillByte := 0, n := SIZEOF(_buf));
            _k3 := _ret.M_StartRead(Key := _M_Key(Name := 'Pool'), pData := ADR(_buf),
                Size := SIZEOF(_buf));
            _s3 := 2;
        END_IF
    2:
        IF _ret.M_Poll(Ticket := _k3, Result := _r3) THEN
            AssertTrue(Condition := _r3.Found AND NOT _r3.Lost, Message := 'and comes back');
            AssertEquals_DINT(Expected := 0, Actual := MEMCMP(pBuf1 := ADR(_buf),
                pBuf2 := ADR(_docB), n := SIZEOF(_docB)), Message := 'byte for byte');
            _k3 := _ret.M_StartWrite(Key := _M_Key(Name := 'Pool'), pData := ADR(_docB), Size := 0);
            _s3 := 3;
        END_IF
    3:
        IF _ret.M_Poll(Ticket := _k3, Result := _r3) THEN
            _k3 := _ret.M_StartRead(Key := _M_Key(Name := 'Pool'), pData := ADR(_buf),
                Size := SIZEOF(_buf));
            _s3 := 4;
        END_IF
    4:
        IF _ret.M_Poll(Ticket := _k3, Result := _r3) THEN
            AssertTrue(Condition := _r3.Ok AND NOT _r3.Found AND NOT _r3.Lost,
                Message := 'an empty document frees the slot');
            _n3 := 1;
            _full3 := 0;
            _s3 := 5;
        END_IF
    5:      // fill the pool until it refuses
        _k3 := _ret.M_StartWrite(Key := _M_Key(Name := CONCAT('Fill', INT_TO_STRING(_n3))),
            pData := ADR(_docA), Size := SIZEOF(_docA));
        _s3 := 6;
    6:
        IF _ret.M_Poll(Ticket := _k3, Result := _r3) THEN
            IF NOT _r3.Ok THEN
                _full3 := _n3;
                AssertEquals_UDINT(Expected := 16#70A, Actual := _r3.ErrorId,
                    Message := 'a full pool refuses with the memory error');
                _n3 := _n3 - 1;
                _s3 := 7;
            ELSIF _n3 > PL_Fraktal.MAX_RETAIN_DOCUMENTS THEN
                AssertTrue(Condition := FALSE, Message := 'the pool took more documents than it holds');
                _s3 := 7;
            ELSE
                _n3 := _n3 + 1;
                _s3 := 5;
            END_IF
        END_IF
    7:      // remove what this run wrote
        IF _n3 < 1 THEN
            AssertTrue(Condition := (_full3 > 0) AND (_full3 <= PL_Fraktal.MAX_RETAIN_DOCUMENTS + 1),
                Message := 'the pool is bounded by MAX_RETAIN_DOCUMENTS');
            _s3 := 99;
            TEST_FINISHED();
        ELSE
            _k3 := _ret.M_StartWrite(Key := _M_Key(Name := CONCAT('Fill', INT_TO_STRING(_n3))),
                pData := ADR(_docA), Size := 0);
            _s3 := 8;
        END_IF
    8:
        IF _ret.M_Poll(Ticket := _k3, Result := _r3) THEN
            _n3 := _n3 - 1;
            _s3 := 7;
        END_IF
    99:
        ;
ELSE
    _s3 := 99;
END_CASE
END_METHOD

